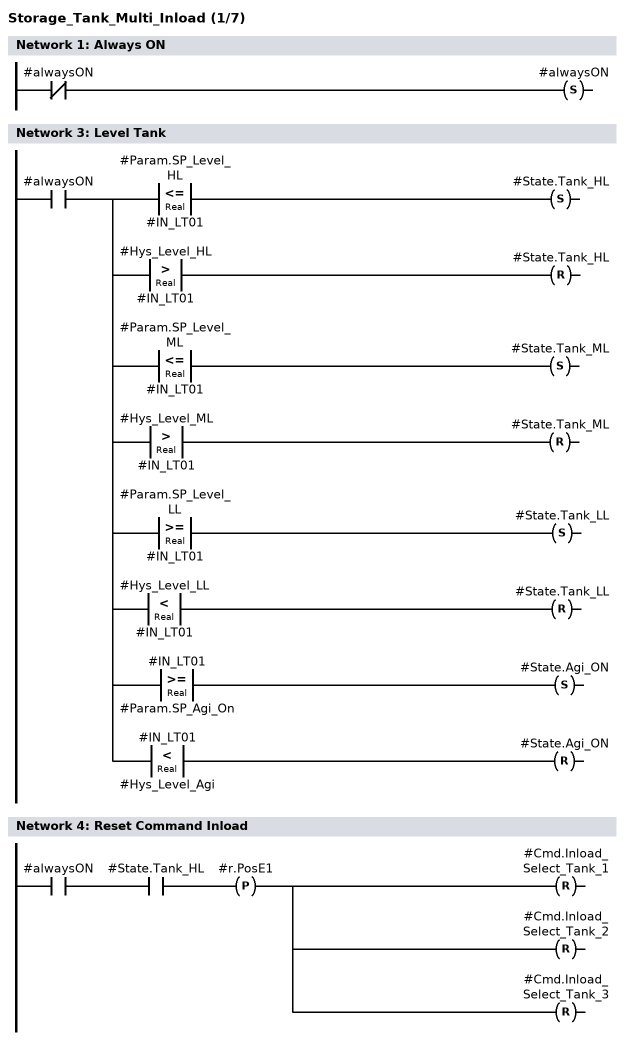
   RUNG wire#powerrail
      I_Contact( #alwaysON )
      S_Coil( #alwaysON )
   END_RUNG
   // the same network as SCL:
   IF NOT #alwaysON THEN #alwaysON := TRUE; END_IF;
END_REGION

NETWORK
TITLE = Hys Calculation
//Level Hys Absolute
      L     #Param.L_Hi_Lim;
      L     #Param.L_Lo_Lim;
      -R;
      L     100.0;
      /R;
      L     #Param.L_Hys;
      *R;
      T     #L_Hys_Abs;
//Tank High Level
      L     #Param.SP_Level_HL;
      L     #L_Hys_Abs;
      -R;
      T     #Hys_Level_HL;
//Tank Mid Level
      L     #Param.SP_Level_ML;
      L     #L_Hys_Abs;
      -R;
      T     #Hys_Level_ML;
//Tank Low Level
      L     #Param.SP_Level_LL;
      L     #L_Hys_Abs;
      +R;
      T     #Hys_Level_LL;
//Level Agi On
      L     #Param.SP_Agi_On;
      L     #L_Hys_Abs;
      -R;
      T     #Hys_Level_Agi;




REGION Network 3: Level Tank
   RUNG wire#powerrail
      Contact( #alwaysON )
      wire#w1
      { S7_Templates := "SrcType := Real" } LE_Contact(in1 := #Param.SP_Level_HL, in2 := #IN_LT01)
      S_Coil( #State.Tank_HL )
   END_RUNG
   RUNG wire#w1
      { S7_Templates := "SrcType := Real" } GT_Contact(in1 := #Hys_Level_HL, in2 := #IN_LT01)
      R_Coil( #State.Tank_HL )
   END_RUNG
   RUNG wire#w1
      { S7_Templates := "SrcType := Real" } LE_Contact(in1 := #Param.SP_Level_ML, in2 := #IN_LT01)
      S_Coil( #State.Tank_ML )
   END_RUNG
   RUNG wire#w1
      { S7_Templates := "SrcType := Real" } GT_Contact(in1 := #Hys_Level_ML, in2 := #IN_LT01)
      R_Coil( #State.Tank_ML )
   END_RUNG
   RUNG wire#w1
      { S7_Templates := "SrcType := Real" } GE_Contact(in1 := #Param.SP_Level_LL, in2 := #IN_LT01)
      S_Coil( #State.Tank_LL )
   END_RUNG
   RUNG wire#w1
      { S7_Templates := "SrcType := Real" } LT_Contact(in1 := #Hys_Level_LL, in2 := #IN_LT01)
      R_Coil( #State.Tank_LL )
   END_RUNG
   RUNG wire#w1
      { S7_Templates := "SrcType := Real" } GE_Contact(in1 := #IN_LT01, in2 := #Param.SP_Agi_On)
      S_Coil( #State.Agi_ON )
   END_RUNG
   RUNG wire#w1
      { S7_Templates := "SrcType := Real" } LT_Contact(in1 := #IN_LT01, in2 := #Hys_Level_Agi)
      R_Coil( #State.Agi_ON )
   END_RUNG
   // the same network as SCL:
   IF #alwaysON AND (#Param.SP_Level_HL <= #IN_LT01) THEN #State.Tank_HL := TRUE; END_IF;
   IF #alwaysON AND (#Hys_Level_HL > #IN_LT01) THEN #State.Tank_HL := FALSE; END_IF;
   IF #alwaysON AND (#Param.SP_Level_ML <= #IN_LT01) THEN #State.Tank_ML := TRUE; END_IF;
   IF #alwaysON AND (#Hys_Level_ML > #IN_LT01) THEN #State.Tank_ML := FALSE; END_IF;
   IF #alwaysON AND (#Param.SP_Level_LL >= #IN_LT01) THEN #State.Tank_LL := TRUE; END_IF;
   IF #alwaysON AND (#Hys_Level_LL < #IN_LT01) THEN #State.Tank_LL := FALSE; END_IF;
   IF #alwaysON AND (#IN_LT01 >= #Param.SP_Agi_On) THEN #State.Agi_ON := TRUE; END_IF;
   IF #alwaysON AND (#IN_LT01 < #Hys_Level_Agi) THEN #State.Agi_ON := FALSE; END_IF;
END_REGION

REGION Network 4: Reset Command Inload
   RUNG wire#powerrail
      Contact( #alwaysON )
      Contact( #State.Tank_HL )
      P_Trig( #r.PosE1 )
      wire#w1
      R_Coil( #Cmd.Inload_Select_Tank_1 )
   END_RUNG
   RUNG wire#w1
      R_Coil( #Cmd.Inload_Select_Tank_2 )
   END_RUNG
   RUNG wire#w1
      R_Coil( #Cmd.Inload_Select_Tank_3 )
   END_RUNG
   // the same network as SCL:
   #_w1 := #alwaysON AND #State.Tank_HL;
   #_w2 := #_w1 AND NOT #r.PosE1;   // rising edge
   #r.PosE1 := #_w1;
   IF #_w2 THEN
       #Cmd.Inload_Select_Tank_1 := FALSE;
       #Cmd.Inload_Select_Tank_2 := FALSE;
       #Cmd.Inload_Select_Tank_3 := FALSE;
   END_IF;
END_REGION

REGION Network 5: Command Inload
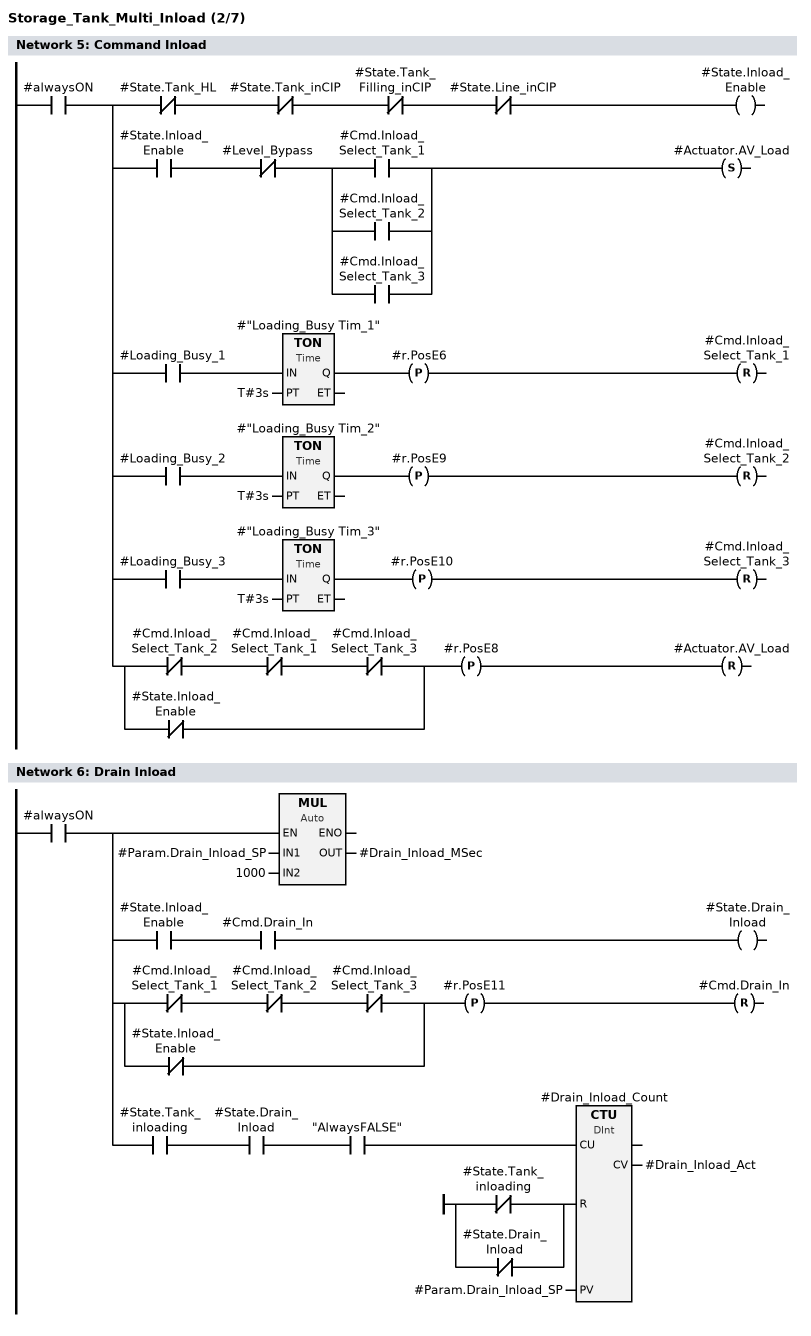
   RUNG wire#powerrail
      Contact( #alwaysON )
      wire#w1
      I_Contact( #State.Tank_HL )
      I_Contact( #State.Tank_inCIP )
      I_Contact( #State.Tank_Filling_inCIP )
      I_Contact( #State.Line_inCIP )
      Coil( #State.Inload_Enable )
   END_RUNG
   RUNG wire#w1
      Contact( #State.Inload_Enable )
      I_Contact( #Level_Bypass )
      wire#w2
      Contact( #Cmd.Inload_Select_Tank_1 )
      wire#w3
      S_Coil( #Actuator.AV_Load )
   END_RUNG
   RUNG wire#w2
      Contact( #Cmd.Inload_Select_Tank_2 )
   END_RUNG wire#w3
   RUNG wire#w2
      Contact( #Cmd.Inload_Select_Tank_3 )
   END_RUNG wire#w3
   RUNG wire#w1
      Contact( #Loading_Busy_1 )
      { S7_Templates := "time_type := Time" } #"Loading_Busy Tim_1".TON(pt := T#3s, et =>)
      P_Trig( #r.PosE6 )
      R_Coil( #Cmd.Inload_Select_Tank_1 )
   END_RUNG
   RUNG wire#w1
      Contact( #Loading_Busy_2 )
      { S7_Templates := "time_type := Time" } #"Loading_Busy Tim_2".TON(pt := T#3s, et =>)
      P_Trig( #r.PosE9 )
      R_Coil( #Cmd.Inload_Select_Tank_2 )
   END_RUNG
   RUNG wire#w1
      Contact( #Loading_Busy_3 )
      { S7_Templates := "time_type := Time" } #"Loading_Busy Tim_3".TON(pt := T#3s, et =>)
      P_Trig( #r.PosE10 )
      R_Coil( #Cmd.Inload_Select_Tank_3 )
   END_RUNG
   RUNG wire#w1
      I_Contact( #Cmd.Inload_Select_Tank_2 )
      I_Contact( #Cmd.Inload_Select_Tank_1 )
      I_Contact( #Cmd.Inload_Select_Tank_3 )
      wire#w4
      P_Trig( #r.PosE8 )
      R_Coil( #Actuator.AV_Load )
   END_RUNG
   RUNG wire#w1
      I_Contact( #State.Inload_Enable )
   END_RUNG wire#w4
   // the same network as SCL:
   #State.Inload_Enable := #alwaysON AND NOT #State.Tank_HL AND NOT #State.Tank_inCIP AND NOT #State.Tank_Filling_inCIP AND NOT #State.Line_inCIP;
   IF #alwaysON AND #State.Inload_Enable AND NOT #Level_Bypass AND (#Cmd.Inload_Select_Tank_1 OR #Cmd.Inload_Select_Tank_2 OR #Cmd.Inload_Select_Tank_3) THEN
       #Actuator.AV_Load := TRUE;
   END_IF;
   #"Loading_Busy Tim_1"(IN := #alwaysON AND #Loading_Busy_1, PT := T#3s);   // TON
   #_w1 := #"Loading_Busy Tim_1".Q AND NOT #r.PosE6;   // rising edge
   #r.PosE6 := #"Loading_Busy Tim_1".Q;
   IF #_w1 THEN #Cmd.Inload_Select_Tank_1 := FALSE; END_IF;
   #"Loading_Busy Tim_2"(IN := #alwaysON AND #Loading_Busy_2, PT := T#3s);   // TON
   #_w2 := #"Loading_Busy Tim_2".Q AND NOT #r.PosE9;   // rising edge
   #r.PosE9 := #"Loading_Busy Tim_2".Q;
   IF #_w2 THEN #Cmd.Inload_Select_Tank_2 := FALSE; END_IF;
   #"Loading_Busy Tim_3"(IN := #alwaysON AND #Loading_Busy_3, PT := T#3s);   // TON
   #_w3 := #"Loading_Busy Tim_3".Q AND NOT #r.PosE10;   // rising edge
   #r.PosE10 := #"Loading_Busy Tim_3".Q;
   IF #_w3 THEN #Cmd.Inload_Select_Tank_3 := FALSE; END_IF;
   #_w4 := #alwaysON AND ((NOT #Cmd.Inload_Select_Tank_2 AND NOT #Cmd.Inload_Select_Tank_1 AND NOT #Cmd.Inload_Select_Tank_3) OR NOT #State.Inload_Enable);
   #_w5 := #_w4 AND NOT #r.PosE8;   // rising edge
   #r.PosE8 := #_w4;
   IF #_w5 THEN #Actuator.AV_Load := FALSE; END_IF;
END_REGION

REGION Network 6: Drain Inload
   RUNG wire#powerrail
      Contact( #alwaysON )
      wire#w1
      Mul(in1 := #Param.Drain_Inload_SP, in2 := 1000, out => #Drain_Inload_MSec)
   END_RUNG
   RUNG wire#w1
      Contact( #State.Inload_Enable )
      Contact( #Cmd.Drain_In )
      Coil( #State.Drain_Inload )
   END_RUNG
   RUNG wire#w1
      I_Contact( #Cmd.Inload_Select_Tank_1 )
      I_Contact( #Cmd.Inload_Select_Tank_2 )
      I_Contact( #Cmd.Inload_Select_Tank_3 )
      wire#w2
      P_Trig( #r.PosE11 )
      R_Coil( #Cmd.Drain_In )
   END_RUNG
   RUNG wire#w1
      I_Contact( #State.Inload_Enable )
   END_RUNG wire#w2
   RUNG wire#w1
      Contact( #State.Tank_inloading )
      Contact( #State.Drain_Inload )
      Contact( "AlwaysFALSE" )
      { S7_Templates := "value_type := DInt" } #Drain_Inload_Count.CTU(r := wire#w3, pv := #Param.Drain_Inload_SP, cv => #Drain_Inload_Act)
   END_RUNG
   RUNG wire#powerrail
      I_Contact( #State.Tank_inloading )
   END_RUNG wire#w3
   RUNG wire#powerrail
      I_Contact( #State.Drain_Inload )
   END_RUNG wire#w3
   // the same network as SCL:
   IF #alwaysON THEN #Drain_Inload_MSec := #Param.Drain_Inload_SP * 1000; END_IF;
   #State.Drain_Inload := #alwaysON AND #State.Inload_Enable AND #Cmd.Drain_In;
   #_w1 := #alwaysON AND ((NOT #Cmd.Inload_Select_Tank_1 AND NOT #Cmd.Inload_Select_Tank_2 AND NOT #Cmd.Inload_Select_Tank_3) OR NOT #State.Inload_Enable);
   #_w2 := #_w1 AND NOT #r.PosE11;   // rising edge
   #r.PosE11 := #_w1;
   IF #_w2 THEN #Cmd.Drain_In := FALSE; END_IF;
   #Drain_Inload_Count.CTU(CU := #alwaysON AND #State.Tank_inloading AND #State.Drain_Inload AND "AlwaysFALSE",
                           R := NOT #State.Tank_inloading OR NOT #State.Drain_Inload,
                           PV := #Param.Drain_Inload_SP,
                           CV => #Drain_Inload_Act);
END_REGION

REGION Network 7: Command Transfer to Filling
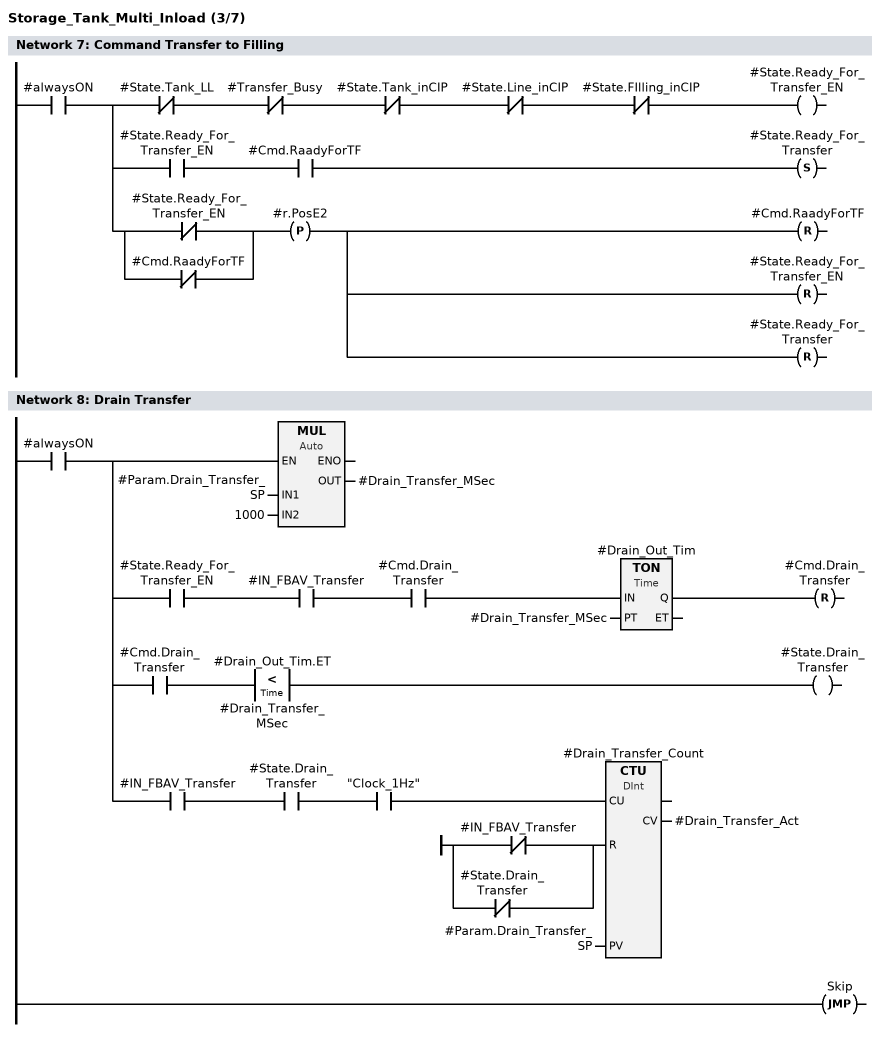
   RUNG wire#powerrail
      Contact( #alwaysON )
      wire#w1
      I_Contact( #State.Tank_LL )
      I_Contact( #Transfer_Busy )
      I_Contact( #State.Tank_inCIP )
      I_Contact( #State.Line_inCIP )
      I_Contact( #State.FIlling_inCIP )
      Coil( #State.Ready_For_Transfer_EN )
   END_RUNG
   RUNG wire#w1
      Contact( #State.Ready_For_Transfer_EN )
      Contact( #Cmd.RaadyForTF )
      S_Coil( #State.Ready_For_Transfer )
   END_RUNG
   RUNG wire#w1
      I_Contact( #State.Ready_For_Transfer_EN )
      wire#w2
      P_Trig( #r.PosE2 )
      wire#w3
      R_Coil( #Cmd.RaadyForTF )
   END_RUNG
   RUNG wire#w1
      I_Contact( #Cmd.RaadyForTF )
   END_RUNG wire#w2
   RUNG wire#w3
      R_Coil( #State.Ready_For_Transfer_EN )
   END_RUNG
   RUNG wire#w3
      R_Coil( #State.Ready_For_Transfer )
   END_RUNG
   // the same network as SCL:
   #State.Ready_For_Transfer_EN := #alwaysON AND NOT #State.Tank_LL AND NOT #Transfer_Busy AND NOT #State.Tank_inCIP AND NOT #State.Line_inCIP AND NOT #State.FIlling_inCIP;
   IF #alwaysON AND #State.Ready_For_Transfer_EN AND #Cmd.RaadyForTF THEN
       #State.Ready_For_Transfer := TRUE;
   END_IF;
   #_w1 := #alwaysON AND (NOT #State.Ready_For_Transfer_EN OR NOT #Cmd.RaadyForTF);
   #_w2 := #_w1 AND NOT #r.PosE2;   // rising edge
   #r.PosE2 := #_w1;
   IF #_w2 THEN
       #Cmd.RaadyForTF := FALSE;
       #State.Ready_For_Transfer_EN := FALSE;
       #State.Ready_For_Transfer := FALSE;
   END_IF;
END_REGION

REGION Network 8: Drain Transfer
   RUNG wire#powerrail
      Contact( #alwaysON )
      wire#w1
      Mul(in1 := #Param.Drain_Transfer_SP, in2 := 1000, out => #Drain_Transfer_MSec)
   END_RUNG
   RUNG wire#w1
      Contact( #State.Ready_For_Transfer_EN )
      Contact( #IN_FBAV_Transfer )
      Contact( #Cmd.Drain_Transfer )
      { S7_Templates := "time_type := Time" } #Drain_Out_Tim.TON(pt := #Drain_Transfer_MSec, et =>)
      R_Coil( #Cmd.Drain_Transfer )
   END_RUNG
   RUNG wire#w1
      Contact( #Cmd.Drain_Transfer )
      { S7_Templates := "SrcType := Time" } LT_Contact(in1 := #Drain_Out_Tim.ET, in2 := #Drain_Transfer_MSec)
      Coil( #State.Drain_Transfer )
   END_RUNG
   RUNG wire#w1
      Contact( #IN_FBAV_Transfer )
      Contact( #State.Drain_Transfer )
      Contact( "Clock_1Hz" )
      { S7_Templates := "value_type := DInt" } #Drain_Transfer_Count.CTU(r := wire#w2, pv := #Param.Drain_Transfer_SP, cv => #Drain_Transfer_Act)
   END_RUNG
   RUNG wire#powerrail
      I_Contact( #IN_FBAV_Transfer )
   END_RUNG wire#w2
   RUNG wire#powerrail
      I_Contact( #State.Drain_Transfer )
   END_RUNG wire#w2
   RUNG wire#powerrail
      JumpCoil( Skip )
   END_RUNG
   // the same network as SCL:
   IF #alwaysON THEN #Drain_Transfer_MSec := #Param.Drain_Transfer_SP * 1000; END_IF;
   #Drain_Out_Tim(IN := #alwaysON AND #State.Ready_For_Transfer_EN AND #IN_FBAV_Transfer AND #Cmd.Drain_Transfer,   // TON
                  PT := #Drain_Transfer_MSec);
   IF #Drain_Out_Tim.Q THEN #Cmd.Drain_Transfer := FALSE; END_IF;
   #State.Drain_Transfer := #alwaysON AND #Cmd.Drain_Transfer AND (#Drain_Out_Tim.ET < #Drain_Transfer_MSec);
   #Drain_Transfer_Count.CTU(CU := #alwaysON AND #IN_FBAV_Transfer AND #State.Drain_Transfer AND "Clock_1Hz",
                           R := NOT #IN_FBAV_Transfer OR NOT #State.Drain_Transfer,
                           PV := #Param.Drain_Transfer_SP,
                           CV => #Drain_Transfer_Act);
   GOTO Skip;
END_REGION

REGION Network 9: -----------------------------------------------State transfer to filling
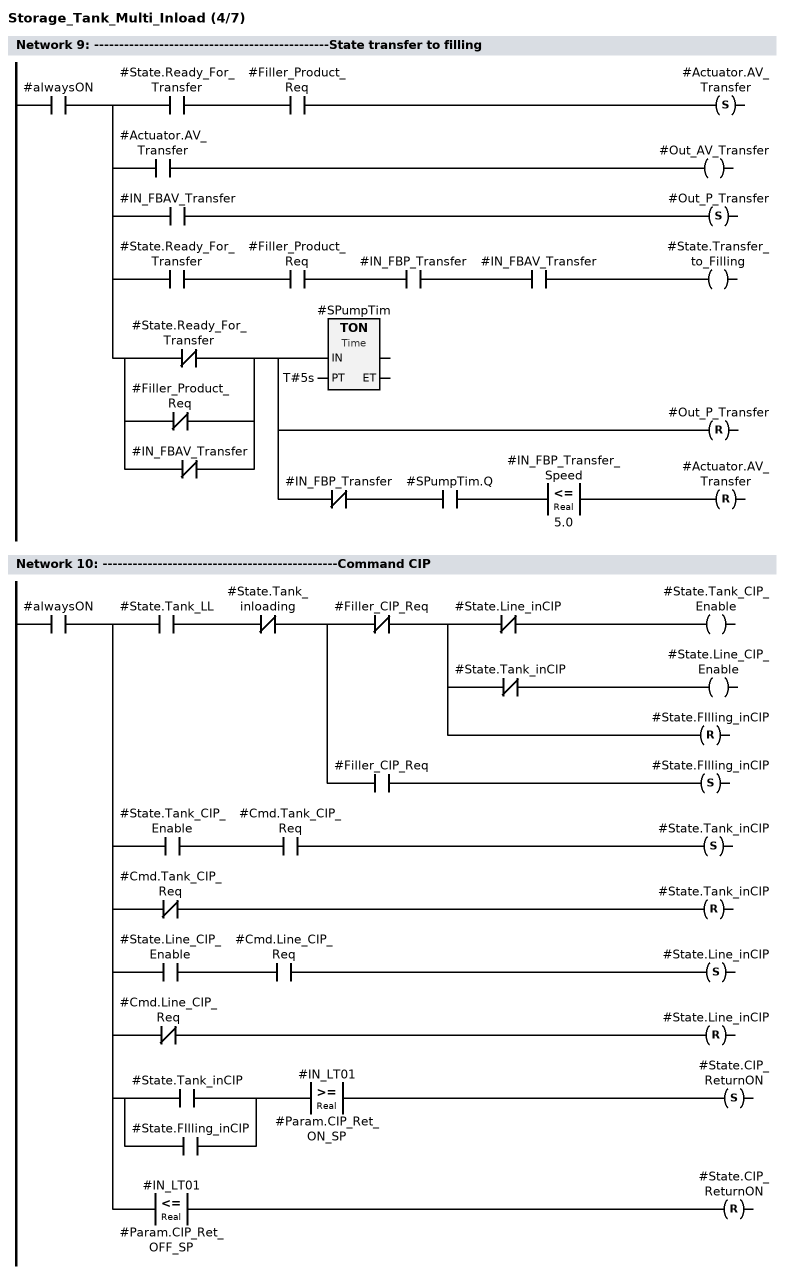
   RUNG wire#powerrail
      Contact( #alwaysON )
      wire#w1
      Contact( #State.Ready_For_Transfer )
      Contact( #Filler_Product_Req )
      S_Coil( #Actuator.AV_Transfer )
   END_RUNG
   RUNG wire#w1
      Contact( #Actuator.AV_Transfer )
      Coil( #Out_AV_Transfer )
   END_RUNG
   RUNG wire#w1
      Contact( #IN_FBAV_Transfer )
      S_Coil( #Out_P_Transfer )
   END_RUNG
   RUNG wire#w1
      Contact( #State.Ready_For_Transfer )
      Contact( #Filler_Product_Req )
      Contact( #IN_FBP_Transfer )
      Contact( #IN_FBAV_Transfer )
      Coil( #State.Transfer_to_Filling )
   END_RUNG
   RUNG wire#w1
      I_Contact( #State.Ready_For_Transfer )
      wire#w2
      { S7_Templates := "time_type := Time" } #SPumpTim.TON(pt := T#5s, et =>)
   END_RUNG
   RUNG wire#w1
      I_Contact( #Filler_Product_Req )
   END_RUNG wire#w2
   RUNG wire#w1
      I_Contact( #IN_FBAV_Transfer )
   END_RUNG wire#w2
   RUNG wire#w2
      R_Coil( #Out_P_Transfer )
   END_RUNG
   RUNG wire#w2
      I_Contact( #IN_FBP_Transfer )
      Contact( #SPumpTim.Q )
      { S7_Templates := "SrcType := Real" } LE_Contact(in1 := #IN_FBP_Transfer_Speed, in2 := 5.0)
      R_Coil( #Actuator.AV_Transfer )
   END_RUNG
   // the same network as SCL:
   IF #alwaysON AND #State.Ready_For_Transfer AND #Filler_Product_Req THEN
       #Actuator.AV_Transfer := TRUE;
   END_IF;
   #Out_AV_Transfer := #alwaysON AND #Actuator.AV_Transfer;
   IF #alwaysON AND #IN_FBAV_Transfer THEN #Out_P_Transfer := TRUE; END_IF;
   #State.Transfer_to_Filling := #alwaysON AND #State.Ready_For_Transfer AND #Filler_Product_Req AND #IN_FBP_Transfer AND #IN_FBAV_Transfer;
   #_w1 := #alwaysON AND (NOT #State.Ready_For_Transfer OR NOT #Filler_Product_Req OR NOT #IN_FBAV_Transfer);
   #SPumpTim(IN := #_w1, PT := T#5s);   // TON
   IF #_w1 THEN #Out_P_Transfer := FALSE; END_IF;
   IF #_w1 AND NOT #IN_FBP_Transfer AND #SPumpTim.Q AND (#IN_FBP_Transfer_Speed <= 5.0) THEN
       #Actuator.AV_Transfer := FALSE;
   END_IF;
END_REGION

REGION Network 10: -----------------------------------------------Command CIP
   RUNG wire#powerrail
      Contact( #alwaysON )
      wire#w1
      Contact( #State.Tank_LL )
      I_Contact( #State.Tank_inloading )
      wire#w2
      I_Contact( #Filler_CIP_Req )
      wire#w3
      I_Contact( #State.Line_inCIP )
      Coil( #State.Tank_CIP_Enable )
   END_RUNG
   RUNG wire#w3
      I_Contact( #State.Tank_inCIP )
      Coil( #State.Line_CIP_Enable )
   END_RUNG
   RUNG wire#w3
      R_Coil( #State.FIlling_inCIP )
   END_RUNG
   RUNG wire#w2
      Contact( #Filler_CIP_Req )
      S_Coil( #State.FIlling_inCIP )
   END_RUNG
   RUNG wire#w1
      Contact( #State.Tank_CIP_Enable )
      Contact( #Cmd.Tank_CIP_Req )
      S_Coil( #State.Tank_inCIP )
   END_RUNG
   RUNG wire#w1
      I_Contact( #Cmd.Tank_CIP_Req )
      R_Coil( #State.Tank_inCIP )
   END_RUNG
   RUNG wire#w1
      Contact( #State.Line_CIP_Enable )
      Contact( #Cmd.Line_CIP_Req )
      S_Coil( #State.Line_inCIP )
   END_RUNG
   RUNG wire#w1
      I_Contact( #Cmd.Line_CIP_Req )
      R_Coil( #State.Line_inCIP )
   END_RUNG
   RUNG wire#w1
      Contact( #State.Tank_inCIP )
      wire#w4
      { S7_Templates := "SrcType := Real" } GE_Contact(in1 := #IN_LT01, in2 := #Param.CIP_Ret_ON_SP)
      S_Coil( #State.CIP_ReturnON )
   END_RUNG
   RUNG wire#w1
      Contact( #State.FIlling_inCIP )
   END_RUNG wire#w4
   RUNG wire#w1
      { S7_Templates := "SrcType := Real" } LE_Contact(in1 := #IN_LT01, in2 := #Param.CIP_Ret_OFF_SP)
      R_Coil( #State.CIP_ReturnON )
   END_RUNG
   // the same network as SCL:
   #_w1 := #alwaysON AND #State.Tank_LL AND NOT #State.Tank_inloading;
   #_w2 := #_w1 AND NOT #Filler_CIP_Req;
   #State.Tank_CIP_Enable := #_w2 AND NOT #State.Line_inCIP;
   #State.Line_CIP_Enable := #_w2 AND NOT #State.Tank_inCIP;
   IF #_w2 THEN #State.FIlling_inCIP := FALSE; END_IF;
   IF #_w1 AND #Filler_CIP_Req THEN #State.FIlling_inCIP := TRUE; END_IF;
   IF #alwaysON AND #State.Tank_CIP_Enable AND #Cmd.Tank_CIP_Req THEN #State.Tank_inCIP := TRUE; END_IF;
   IF #alwaysON AND NOT #Cmd.Tank_CIP_Req THEN #State.Tank_inCIP := FALSE; END_IF;
   IF #alwaysON AND #State.Line_CIP_Enable AND #Cmd.Line_CIP_Req THEN #State.Line_inCIP := TRUE; END_IF;
   IF #alwaysON AND NOT #Cmd.Line_CIP_Req THEN #State.Line_inCIP := FALSE; END_IF;
   IF #alwaysON AND (#State.Tank_inCIP OR #State.FIlling_inCIP) AND (#IN_LT01 >= #Param.CIP_Ret_ON_SP) THEN
       #State.CIP_ReturnON := TRUE;
   END_IF;
   IF #alwaysON AND (#IN_LT01 <= #Param.CIP_Ret_OFF_SP) THEN #State.CIP_ReturnON := FALSE; END_IF;
END_REGION

REGION Network 11: Command CIP New
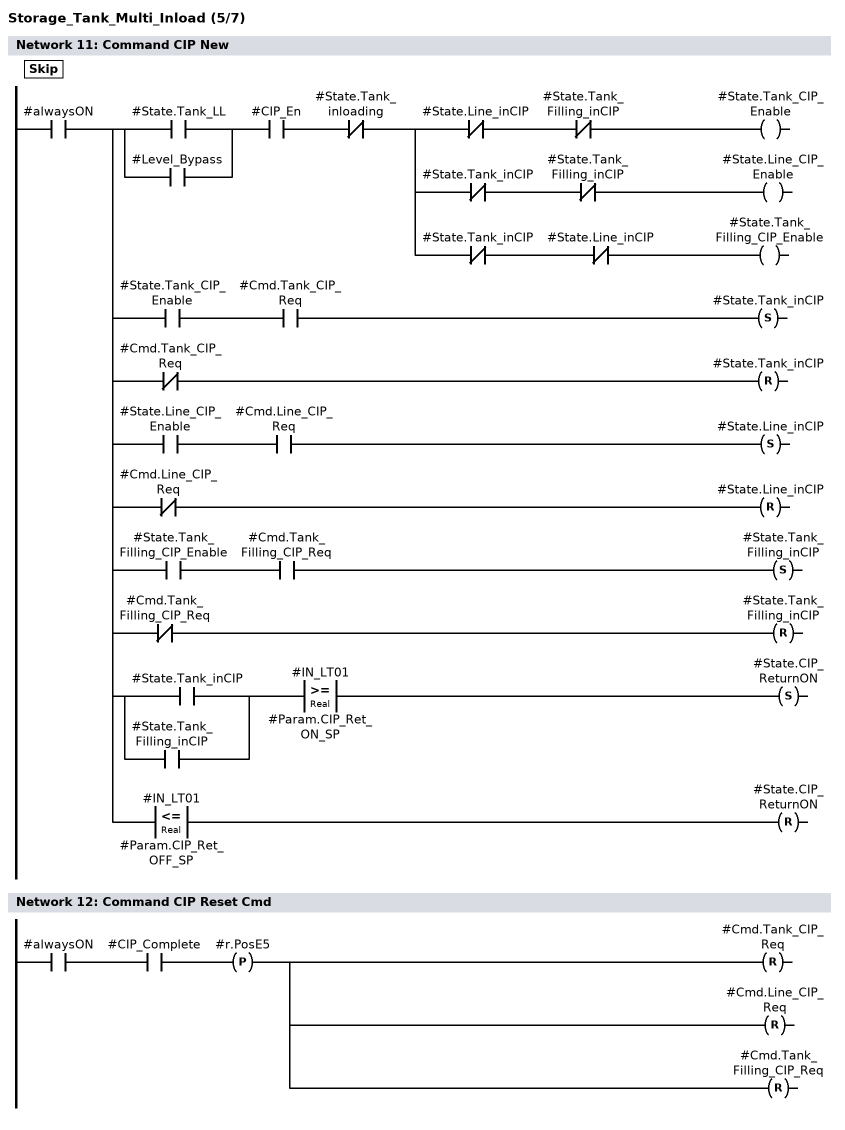
   Label( Skip )
   RUNG wire#powerrail
      Contact( #alwaysON )
      wire#w1
      Contact( #State.Tank_LL )
      wire#w2
      Contact( #CIP_En )
      I_Contact( #State.Tank_inloading )
      wire#w3
      I_Contact( #State.Line_inCIP )
      I_Contact( #State.Tank_Filling_inCIP )
      Coil( #State.Tank_CIP_Enable )
   END_RUNG
   RUNG wire#w1
      Contact( #Level_Bypass )
   END_RUNG wire#w2
   RUNG wire#w3
      I_Contact( #State.Tank_inCIP )
      I_Contact( #State.Tank_Filling_inCIP )
      Coil( #State.Line_CIP_Enable )
   END_RUNG
   RUNG wire#w3
      I_Contact( #State.Tank_inCIP )
      I_Contact( #State.Line_inCIP )
      Coil( #State.Tank_Filling_CIP_Enable )
   END_RUNG
   RUNG wire#w1
      Contact( #State.Tank_CIP_Enable )
      Contact( #Cmd.Tank_CIP_Req )
      S_Coil( #State.Tank_inCIP )
   END_RUNG
   RUNG wire#w1
      I_Contact( #Cmd.Tank_CIP_Req )
      R_Coil( #State.Tank_inCIP )
   END_RUNG
   RUNG wire#w1
      Contact( #State.Line_CIP_Enable )
      Contact( #Cmd.Line_CIP_Req )
      S_Coil( #State.Line_inCIP )
   END_RUNG
   RUNG wire#w1
      I_Contact( #Cmd.Line_CIP_Req )
      R_Coil( #State.Line_inCIP )
   END_RUNG
   RUNG wire#w1
      Contact( #State.Tank_Filling_CIP_Enable )
      Contact( #Cmd.Tank_Filling_CIP_Req )
      S_Coil( #State.Tank_Filling_inCIP )
   END_RUNG
   RUNG wire#w1
      I_Contact( #Cmd.Tank_Filling_CIP_Req )
      R_Coil( #State.Tank_Filling_inCIP )
   END_RUNG
   RUNG wire#w1
      Contact( #State.Tank_inCIP )
      wire#w4
      { S7_Templates := "SrcType := Real" } GE_Contact(in1 := #IN_LT01, in2 := #Param.CIP_Ret_ON_SP)
      S_Coil( #State.CIP_ReturnON )
   END_RUNG
   RUNG wire#w1
      Contact( #State.Tank_Filling_inCIP )
   END_RUNG wire#w4
   RUNG wire#w1
      { S7_Templates := "SrcType := Real" } LE_Contact(in1 := #IN_LT01, in2 := #Param.CIP_Ret_OFF_SP)
      R_Coil( #State.CIP_ReturnON )
   END_RUNG
   // the same network as SCL:
   Skip:
   #_w1 := #alwaysON AND (#State.Tank_LL OR #Level_Bypass) AND #CIP_En AND NOT #State.Tank_inloading;
   #State.Tank_CIP_Enable := #_w1 AND NOT #State.Line_inCIP AND NOT #State.Tank_Filling_inCIP;
   #State.Line_CIP_Enable := #_w1 AND NOT #State.Tank_inCIP AND NOT #State.Tank_Filling_inCIP;
   #State.Tank_Filling_CIP_Enable := #_w1 AND NOT #State.Tank_inCIP AND NOT #State.Line_inCIP;
   IF #alwaysON AND #State.Tank_CIP_Enable AND #Cmd.Tank_CIP_Req THEN #State.Tank_inCIP := TRUE; END_IF;
   IF #alwaysON AND NOT #Cmd.Tank_CIP_Req THEN #State.Tank_inCIP := FALSE; END_IF;
   IF #alwaysON AND #State.Line_CIP_Enable AND #Cmd.Line_CIP_Req THEN #State.Line_inCIP := TRUE; END_IF;
   IF #alwaysON AND NOT #Cmd.Line_CIP_Req THEN #State.Line_inCIP := FALSE; END_IF;
   IF #alwaysON AND #State.Tank_Filling_CIP_Enable AND #Cmd.Tank_Filling_CIP_Req THEN
       #State.Tank_Filling_inCIP := TRUE;
   END_IF;
   IF #alwaysON AND NOT #Cmd.Tank_Filling_CIP_Req THEN #State.Tank_Filling_inCIP := FALSE; END_IF;
   IF #alwaysON AND (#State.Tank_inCIP OR #State.Tank_Filling_inCIP) AND (#IN_LT01 >= #Param.CIP_Ret_ON_SP) THEN
       #State.CIP_ReturnON := TRUE;
   END_IF;
   IF #alwaysON AND (#IN_LT01 <= #Param.CIP_Ret_OFF_SP) THEN #State.CIP_ReturnON := FALSE; END_IF;
END_REGION

REGION Network 12: Command CIP Reset Cmd
   RUNG wire#powerrail
      Contact( #alwaysON )
      Contact( #CIP_Complete )
      P_Trig( #r.PosE5 )
      wire#w1
      R_Coil( #Cmd.Tank_CIP_Req )
   END_RUNG
   RUNG wire#w1
      R_Coil( #Cmd.Line_CIP_Req )
   END_RUNG
   RUNG wire#w1
      R_Coil( #Cmd.Tank_Filling_CIP_Req )
   END_RUNG
   // the same network as SCL:
   #_w1 := #alwaysON AND #CIP_Complete;
   #_w2 := #_w1 AND NOT #r.PosE5;   // rising edge
   #r.PosE5 := #_w1;
   IF #_w2 THEN
       #Cmd.Tank_CIP_Req := FALSE;
       #Cmd.Line_CIP_Req := FALSE;
       #Cmd.Tank_Filling_CIP_Req := FALSE;
   END_IF;
END_REGION

REGION Network 13: Send CIP Request
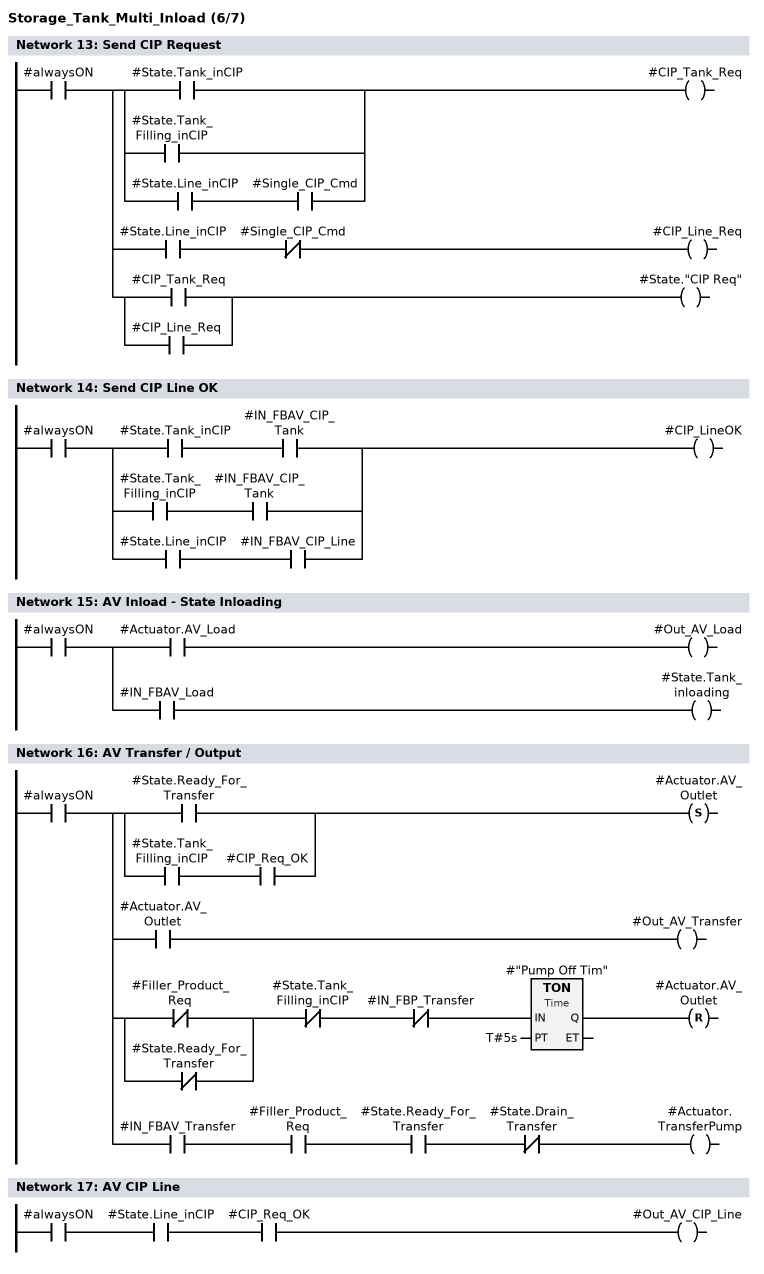
   RUNG wire#powerrail
      Contact( #alwaysON )
      wire#w1
      Contact( #State.Tank_inCIP )
      wire#w2
      Coil( #CIP_Tank_Req )
   END_RUNG
   RUNG wire#w1
      Contact( #State.Tank_Filling_inCIP )
   END_RUNG wire#w2
   RUNG wire#w1
      Contact( #State.Line_inCIP )
      Contact( #Single_CIP_Cmd )
   END_RUNG wire#w2
   RUNG wire#w1
      Contact( #State.Line_inCIP )
      I_Contact( #Single_CIP_Cmd )
      Coil( #CIP_Line_Req )
   END_RUNG
   RUNG wire#w1
      Contact( #CIP_Tank_Req )
      wire#w3
      Coil( #State."CIP Req" )
   END_RUNG
   RUNG wire#w1
      Contact( #CIP_Line_Req )
   END_RUNG wire#w3
   // the same network as SCL:
   #CIP_Tank_Req := #alwaysON AND (#State.Tank_inCIP OR #State.Tank_Filling_inCIP OR (#State.Line_inCIP AND #Single_CIP_Cmd));
   #CIP_Line_Req := #alwaysON AND #State.Line_inCIP AND NOT #Single_CIP_Cmd;
   #State."CIP Req" := #alwaysON AND (#CIP_Tank_Req OR #CIP_Line_Req);
END_REGION

REGION Network 14: Send CIP Line OK
   RUNG wire#powerrail
      Contact( #alwaysON )
      wire#w1
      Contact( #State.Tank_inCIP )
      Contact( #IN_FBAV_CIP_Tank )
      wire#w2
      Coil( #CIP_LineOK )
   END_RUNG
   RUNG wire#w1
      Contact( #State.Tank_Filling_inCIP )
      Contact( #IN_FBAV_CIP_Tank )
   END_RUNG wire#w2
   RUNG wire#w1
      Contact( #State.Line_inCIP )
      Contact( #IN_FBAV_CIP_Line )
   END_RUNG wire#w2
   // the same network as SCL:
   #CIP_LineOK := #alwaysON AND ((#State.Tank_inCIP AND #IN_FBAV_CIP_Tank) OR (#State.Tank_Filling_inCIP AND #IN_FBAV_CIP_Tank) OR (#State.Line_inCIP AND #IN_FBAV_CIP_Line));
END_REGION

REGION Network 15: AV Inload - State Inloading
   RUNG wire#powerrail
      Contact( #alwaysON )
      wire#w1
      Contact( #Actuator.AV_Load )
      Coil( #Out_AV_Load )
   END_RUNG
   RUNG wire#w1
      Contact( #IN_FBAV_Load )
      Coil( #State.Tank_inloading )
   END_RUNG
   // the same network as SCL:
   #Out_AV_Load := #alwaysON AND #Actuator.AV_Load;
   #State.Tank_inloading := #alwaysON AND #IN_FBAV_Load;
END_REGION

REGION Network 16: AV Transfer / Output
   RUNG wire#powerrail
      Contact( #alwaysON )
      wire#w1
      Contact( #State.Ready_For_Transfer )
      wire#w2
      S_Coil( #Actuator.AV_Outlet )
   END_RUNG
   RUNG wire#w1
      Contact( #State.Tank_Filling_inCIP )
      Contact( #CIP_Req_OK )
   END_RUNG wire#w2
   RUNG wire#w1
      Contact( #Actuator.AV_Outlet )
      Coil( #Out_AV_Transfer )
   END_RUNG
   RUNG wire#w1
      I_Contact( #Filler_Product_Req )
      wire#w3
      I_Contact( #State.Tank_Filling_inCIP )
      I_Contact( #IN_FBP_Transfer )
      { S7_Templates := "time_type := Time" } #"Pump Off Tim".TON(pt := T#5s, et =>)
      R_Coil( #Actuator.AV_Outlet )
   END_RUNG
   RUNG wire#w1
      I_Contact( #State.Ready_For_Transfer )
   END_RUNG wire#w3
   RUNG wire#w1
      Contact( #IN_FBAV_Transfer )
      Contact( #Filler_Product_Req )
      Contact( #State.Ready_For_Transfer )
      I_Contact( #State.Drain_Transfer )
      Coil( #Actuator.TransferPump )
   END_RUNG
   // the same network as SCL:
   IF #alwaysON AND (#State.Ready_For_Transfer OR (#State.Tank_Filling_inCIP AND #CIP_Req_OK)) THEN
       #Actuator.AV_Outlet := TRUE;
   END_IF;
   #Out_AV_Transfer := #alwaysON AND #Actuator.AV_Outlet;
   #"Pump Off Tim"(IN := #alwaysON AND (NOT #Filler_Product_Req OR NOT #State.Ready_For_Transfer) AND NOT #State.Tank_Filling_inCIP AND NOT #IN_FBP_Transfer,   // TON
                   PT := T#5s);
   IF #"Pump Off Tim".Q THEN #Actuator.AV_Outlet := FALSE; END_IF;
   #Actuator.TransferPump := #alwaysON AND #IN_FBAV_Transfer AND #Filler_Product_Req AND #State.Ready_For_Transfer AND NOT #State.Drain_Transfer;
END_REGION

REGION Network 17: AV CIP Line
   RUNG wire#powerrail
      Contact( #alwaysON )
      Contact( #State.Line_inCIP )
      Contact( #CIP_Req_OK )
      Coil( #Out_AV_CIP_Line )
   END_RUNG
   // the same network as SCL:
   #Out_AV_CIP_Line := #alwaysON AND #State.Line_inCIP AND #CIP_Req_OK;
END_REGION

REGION Network 18: AV CIP Tank to Filling
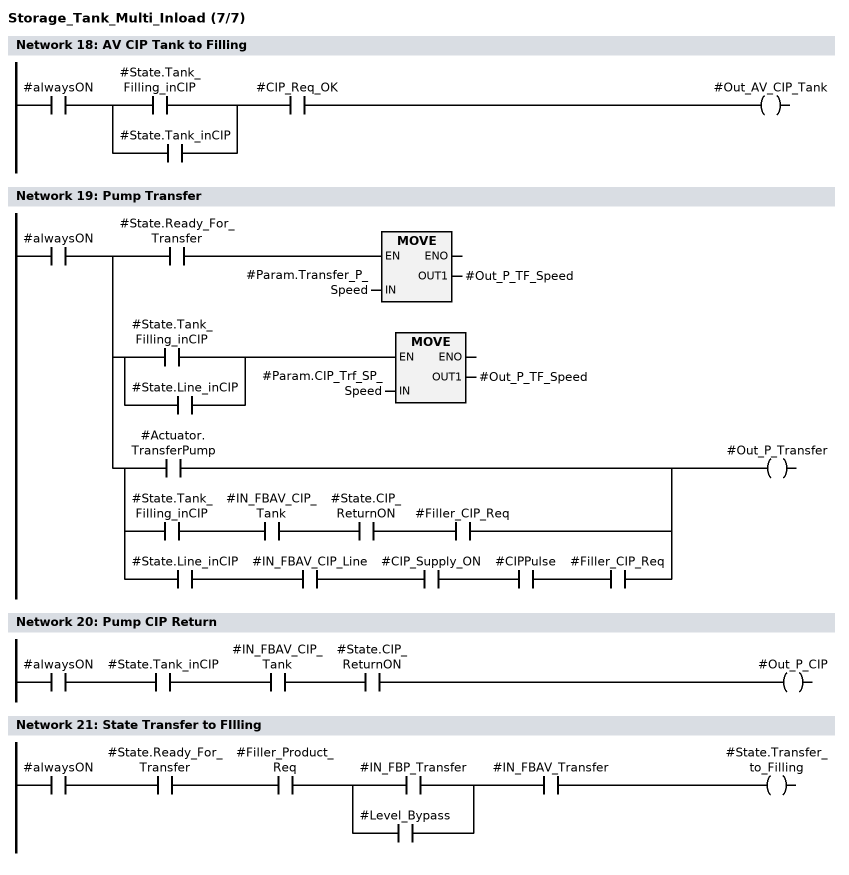
   RUNG wire#powerrail
      Contact( #alwaysON )
      wire#w1
      Contact( #State.Tank_Filling_inCIP )
      wire#w2
      Contact( #CIP_Req_OK )
      Coil( #Out_AV_CIP_Tank )
   END_RUNG
   RUNG wire#w1
      Contact( #State.Tank_inCIP )
   END_RUNG wire#w2
   // the same network as SCL:
   #Out_AV_CIP_Tank := #alwaysON AND (#State.Tank_Filling_inCIP OR #State.Tank_inCIP) AND #CIP_Req_OK;
END_REGION

REGION Network 19: Pump Transfer
   RUNG wire#powerrail
      Contact( #alwaysON )
      wire#w1
      Contact( #State.Ready_For_Transfer )
      Move(in := #Param.Transfer_P_Speed, out1 => #Out_P_TF_Speed)
   END_RUNG
   RUNG wire#w1
      Contact( #State.Tank_Filling_inCIP )
      wire#w2
      Move(in := #Param.CIP_Trf_SP_Speed, out1 => #Out_P_TF_Speed)
   END_RUNG
   RUNG wire#w1
      Contact( #State.Line_inCIP )
   END_RUNG wire#w2
   RUNG wire#w1
      Contact( #Actuator.TransferPump )
      wire#w3
      Coil( #Out_P_Transfer )
   END_RUNG
   RUNG wire#w1
      Contact( #State.Tank_Filling_inCIP )
      Contact( #IN_FBAV_CIP_Tank )
      Contact( #State.CIP_ReturnON )
      Contact( #Filler_CIP_Req )
   END_RUNG wire#w3
   RUNG wire#w1
      Contact( #State.Line_inCIP )
      Contact( #IN_FBAV_CIP_Line )
      Contact( #CIP_Supply_ON )
      Contact( #CIPPulse )
      Contact( #Filler_CIP_Req )
   END_RUNG wire#w3
   // the same network as SCL:
   IF #alwaysON AND #State.Ready_For_Transfer THEN #Out_P_TF_Speed := #Param.Transfer_P_Speed; END_IF;
   IF #alwaysON AND (#State.Tank_Filling_inCIP OR #State.Line_inCIP) THEN
       #Out_P_TF_Speed := #Param.CIP_Trf_SP_Speed;
   END_IF;
   #Out_P_Transfer := #alwaysON AND (#Actuator.TransferPump OR (#State.Tank_Filling_inCIP AND #IN_FBAV_CIP_Tank AND #State.CIP_ReturnON AND #Filler_CIP_Req) OR (#State.Line_inCIP AND #IN_FBAV_CIP_Line AND #CIP_Supply_ON AND #CIPPulse AND #Filler_CIP_Req));
END_REGION

REGION Network 20: Pump CIP Return
   RUNG wire#powerrail
      Contact( #alwaysON )
      Contact( #State.Tank_inCIP )
      Contact( #IN_FBAV_CIP_Tank )
      Contact( #State.CIP_ReturnON )
      Coil( #Out_P_CIP )
   END_RUNG
   // the same network as SCL:
   #Out_P_CIP := #alwaysON AND #State.Tank_inCIP AND #IN_FBAV_CIP_Tank AND #State.CIP_ReturnON;
END_REGION

REGION Network 21: State Transfer to FIlling
   RUNG wire#powerrail
      Contact( #alwaysON )
      Contact( #State.Ready_For_Transfer )
      Contact( #Filler_Product_Req )
      wire#w1
      Contact( #IN_FBP_Transfer )
      wire#w2
      Contact( #IN_FBAV_Transfer )
      Coil( #State.Transfer_to_Filling )
   END_RUNG
   RUNG wire#w1
      Contact( #Level_Bypass )
   END_RUNG wire#w2
   // the same network as SCL:
   #State.Transfer_to_Filling := #alwaysON AND #State.Ready_For_Transfer AND #Filler_Product_Req AND (#IN_FBP_Transfer OR #Level_Bypass) AND #IN_FBAV_Transfer;
END_REGION
END_FUNCTION_BLOCK

FUNCTION "Buffer" : Void   // FC11, LAD
{ S7_Optimized_Access := 'TRUE' }
VERSION : 0.1
// stored: AutoNumber true, IsIECCheckEnabled false, SetENOAutomatically false, UDAEnableTagReadback false
BEGIN

REGION Network 1: BFT 61 Rework 32
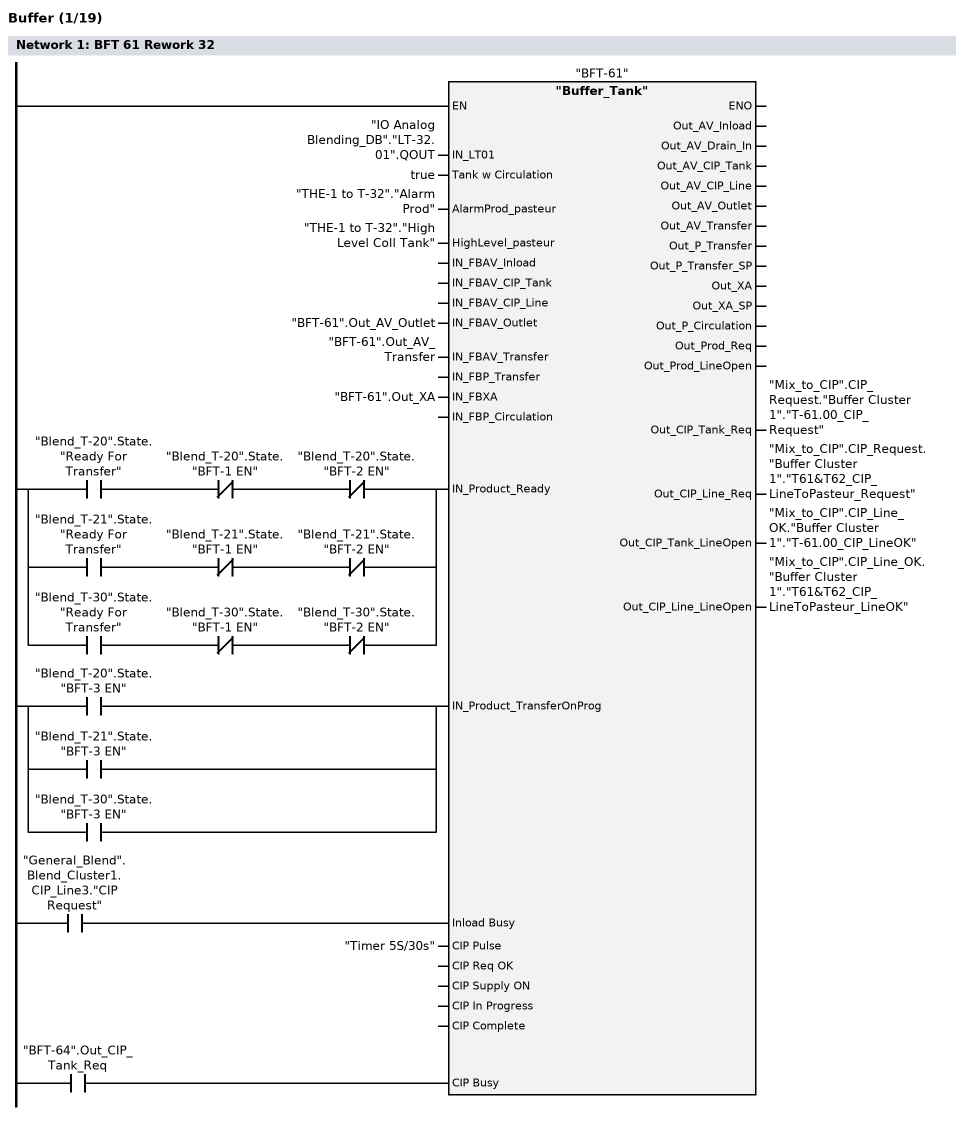
   RUNG wire#powerrail
      "BFT-61"(IN_Product_Ready := wire#w1, IN_Product_TransferOnProg := wire#w2, "Inload Busy" := wire#w3, "CIP Busy" := wire#w4, IN_LT01 := "IO Analog Blending_DB"."LT-32.01".QOUT, "Tank w Circulation" := true, AlarmProd_pasteur := "THE-1 to T-32"."Alarm Prod", HighLevel_pasteur := "THE-1 to T-32"."High Level Coll Tank", IN_FBAV_Inload :=, IN_FBAV_CIP_Tank :=, IN_FBAV_CIP_Line :=, IN_FBAV_Outlet := "BFT-61".Out_AV_Outlet, IN_FBAV_Transfer := "BFT-61".Out_AV_Transfer, IN_FBP_Transfer :=, IN_FBXA := "BFT-61".Out_XA, IN_FBP_Circulation :=, "CIP Pulse" := "Timer 5S/30s", "CIP Req OK" :=, "CIP Supply ON" :=, "CIP In Progress" :=, "CIP Complete" :=, Out_AV_Inload =>, Out_AV_Drain_In =>, Out_AV_CIP_Tank =>, Out_AV_CIP_Line =>, Out_AV_Outlet =>, Out_AV_Transfer =>, Out_P_Transfer =>, Out_P_Transfer_SP =>, Out_XA =>, Out_XA_SP =>, Out_P_Circulation =>, Out_Prod_Req =>, Out_Prod_LineOpen =>, Out_CIP_Tank_Req => "Mix_to_CIP".CIP_Request."Buffer Cluster 1"."T-61.00_CIP_Request", Out_CIP_Line_Req => "Mix_to_CIP".CIP_Request."Buffer Cluster 1"."T61&T62_CIP_LineToPasteur_Request", Out_CIP_Tank_LineOpen => "Mix_to_CIP".CIP_Line_OK."Buffer Cluster 1"."T-61.00_CIP_LineOK", Out_CIP_Line_LineOpen => "Mix_to_CIP".CIP_Line_OK."Buffer Cluster 1"."T61&T62_CIP_LineToPasteur_LineOK")
   END_RUNG
   RUNG wire#powerrail
      Contact( "Blend_T-20".State."Ready For Transfer" )
      I_Contact( "Blend_T-20".State."BFT-1 EN" )
      I_Contact( "Blend_T-20".State."BFT-2 EN" )
   END_RUNG wire#w1
   RUNG wire#powerrail
      Contact( "Blend_T-21".State."Ready For Transfer" )
      I_Contact( "Blend_T-21".State."BFT-1 EN" )
      I_Contact( "Blend_T-21".State."BFT-2 EN" )
   END_RUNG wire#w1
   RUNG wire#powerrail
      Contact( "Blend_T-30".State."Ready For Transfer" )
      I_Contact( "Blend_T-30".State."BFT-1 EN" )
      I_Contact( "Blend_T-30".State."BFT-2 EN" )
   END_RUNG wire#w1
   RUNG wire#powerrail
      Contact( "Blend_T-20".State."BFT-3 EN" )
   END_RUNG wire#w2
   RUNG wire#powerrail
      Contact( "Blend_T-21".State."BFT-3 EN" )
   END_RUNG wire#w2
   RUNG wire#powerrail
      Contact( "Blend_T-30".State."BFT-3 EN" )
   END_RUNG wire#w2
   RUNG wire#powerrail
      Contact( "General_Blend".Blend_Cluster1.CIP_Line3."CIP Request" )
   END_RUNG wire#w3
   RUNG wire#powerrail
      Contact( "BFT-64".Out_CIP_Tank_Req )
   END_RUNG wire#w4
   // the same network as SCL:
   "BFT-61"(IN_LT01 := "IO Analog Blending_DB"."LT-32.01".QOUT,   // "Buffer_Tank"
            "Tank w Circulation" := true,
            AlarmProd_pasteur := "THE-1 to T-32"."Alarm Prod",
            HighLevel_pasteur := "THE-1 to T-32"."High Level Coll Tank",
            IN_FBAV_Outlet := "BFT-61".Out_AV_Outlet,
            IN_FBAV_Transfer := "BFT-61".Out_AV_Transfer,
            IN_FBXA := "BFT-61".Out_XA,
            IN_Product_Ready := ("Blend_T-20".State."Ready For Transfer" AND NOT "Blend_T-20".State."BFT-1 EN" AND NOT "Blend_T-20".State."BFT-2 EN") OR ("Blend_T-21".State."Ready For Transfer" AND NOT "Blend_T-21".State."BFT-1 EN" AND NOT "Blend_T-21".State."BFT-2 EN") OR ("Blend_T-30".State."Ready For Transfer" AND NOT "Blend_T-30".State."BFT-1 EN" AND NOT "Blend_T-30".State."BFT-2 EN"),
            IN_Product_TransferOnProg := "Blend_T-20".State."BFT-3 EN" OR "Blend_T-21".State."BFT-3 EN" OR "Blend_T-30".State."BFT-3 EN",
            "Inload Busy" := "General_Blend".Blend_Cluster1.CIP_Line3."CIP Request",
            "CIP Pulse" := "Timer 5S/30s",
            "CIP Busy" := "BFT-64".Out_CIP_Tank_Req,
            Out_CIP_Tank_Req => "Mix_to_CIP".CIP_Request."Buffer Cluster 1"."T-61.00_CIP_Request",
            Out_CIP_Line_Req => "Mix_to_CIP".CIP_Request."Buffer Cluster 1"."T61&T62_CIP_LineToPasteur_Request",
            Out_CIP_Tank_LineOpen => "Mix_to_CIP".CIP_Line_OK."Buffer Cluster 1"."T-61.00_CIP_LineOK",
            Out_CIP_Line_LineOpen => "Mix_to_CIP".CIP_Line_OK."Buffer Cluster 1"."T61&T62_CIP_LineToPasteur_LineOK");
END_REGION

REGION Network 2: BFT 61 Feedback Instrument
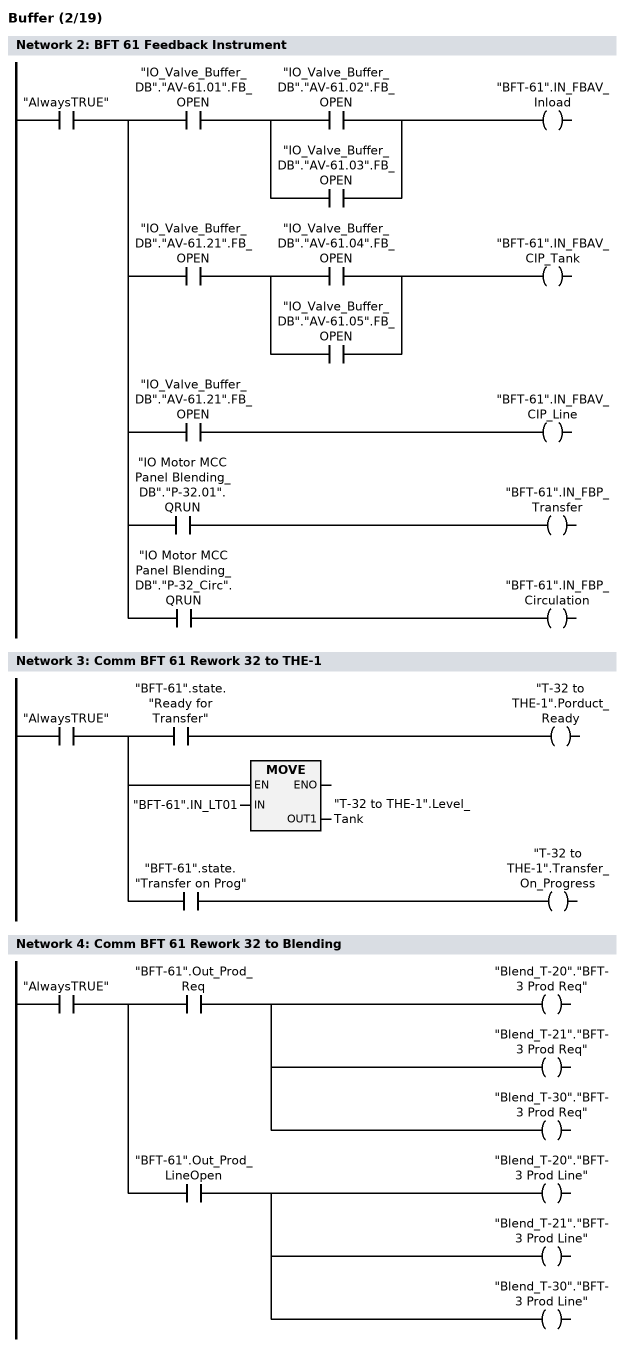
   RUNG wire#powerrail
      Contact( "AlwaysTRUE" )
      wire#w1
      Contact( "IO_Valve_Buffer_DB"."AV-61.01".FB_OPEN )
      wire#w2
      Contact( "IO_Valve_Buffer_DB"."AV-61.02".FB_OPEN )
      wire#w3
      Coil( "BFT-61".IN_FBAV_Inload )
   END_RUNG
   RUNG wire#w2
      Contact( "IO_Valve_Buffer_DB"."AV-61.03".FB_OPEN )
   END_RUNG wire#w3
   RUNG wire#w1
      Contact( "IO_Valve_Buffer_DB"."AV-61.21".FB_OPEN )
      wire#w4
      Contact( "IO_Valve_Buffer_DB"."AV-61.04".FB_OPEN )
      wire#w5
      Coil( "BFT-61".IN_FBAV_CIP_Tank )
   END_RUNG
   RUNG wire#w4
      Contact( "IO_Valve_Buffer_DB"."AV-61.05".FB_OPEN )
   END_RUNG wire#w5
   RUNG wire#w1
      Contact( "IO_Valve_Buffer_DB"."AV-61.21".FB_OPEN )
      Coil( "BFT-61".IN_FBAV_CIP_Line )
   END_RUNG
   RUNG wire#w1
      Contact( "IO Motor MCC Panel Blending_DB"."P-32.01".QRUN )
      Coil( "BFT-61".IN_FBP_Transfer )
   END_RUNG
   RUNG wire#w1
      Contact( "IO Motor MCC Panel Blending_DB"."P-32_Circ".QRUN )
      Coil( "BFT-61".IN_FBP_Circulation )
   END_RUNG
   // the same network as SCL:
   "BFT-61".IN_FBAV_Inload := "AlwaysTRUE" AND "IO_Valve_Buffer_DB"."AV-61.01".FB_OPEN AND ("IO_Valve_Buffer_DB"."AV-61.02".FB_OPEN OR "IO_Valve_Buffer_DB"."AV-61.03".FB_OPEN);
   "BFT-61".IN_FBAV_CIP_Tank := "AlwaysTRUE" AND "IO_Valve_Buffer_DB"."AV-61.21".FB_OPEN AND ("IO_Valve_Buffer_DB"."AV-61.04".FB_OPEN OR "IO_Valve_Buffer_DB"."AV-61.05".FB_OPEN);
   "BFT-61".IN_FBAV_CIP_Line := "AlwaysTRUE" AND "IO_Valve_Buffer_DB"."AV-61.21".FB_OPEN;
   "BFT-61".IN_FBP_Transfer := "AlwaysTRUE" AND "IO Motor MCC Panel Blending_DB"."P-32.01".QRUN;
   "BFT-61".IN_FBP_Circulation := "AlwaysTRUE" AND "IO Motor MCC Panel Blending_DB"."P-32_Circ".QRUN;
END_REGION

REGION Network 3: Comm BFT 61 Rework 32 to THE-1
   RUNG wire#powerrail
      Contact( "AlwaysTRUE" )
      wire#w1
      Contact( "BFT-61".state."Ready for Transfer" )
      Coil( "T-32 to THE-1".Porduct_Ready )
   END_RUNG
   RUNG wire#w1
      Move(in := "BFT-61".IN_LT01, out1 => "T-32 to THE-1".Level_Tank)
   END_RUNG
   RUNG wire#w1
      Contact( "BFT-61".state."Transfer on Prog" )
      Coil( "T-32 to THE-1".Transfer_On_Progress )
   END_RUNG
   // the same network as SCL:
   "T-32 to THE-1".Porduct_Ready := "AlwaysTRUE" AND "BFT-61".state."Ready for Transfer";
   IF "AlwaysTRUE" THEN "T-32 to THE-1".Level_Tank := "BFT-61".IN_LT01; END_IF;
   "T-32 to THE-1".Transfer_On_Progress := "AlwaysTRUE" AND "BFT-61".state."Transfer on Prog";
END_REGION

REGION Network 4: Comm BFT 61 Rework 32 to Blending
   RUNG wire#powerrail
      Contact( "AlwaysTRUE" )
      wire#w1
      Contact( "BFT-61".Out_Prod_Req )
      wire#w2
      Coil( "Blend_T-20"."BFT-3 Prod Req" )
   END_RUNG
   RUNG wire#w2
      Coil( "Blend_T-21"."BFT-3 Prod Req" )
   END_RUNG
   RUNG wire#w2
      Coil( "Blend_T-30"."BFT-3 Prod Req" )
   END_RUNG
   RUNG wire#w1
      Contact( "BFT-61".Out_Prod_LineOpen )
      wire#w3
      Coil( "Blend_T-20"."BFT-3 Prod Line" )
   END_RUNG
   RUNG wire#w3
      Coil( "Blend_T-21"."BFT-3 Prod Line" )
   END_RUNG
   RUNG wire#w3
      Coil( "Blend_T-30"."BFT-3 Prod Line" )
   END_RUNG
   // the same network as SCL:
   "Blend_T-20"."BFT-3 Prod Req" := "AlwaysTRUE" AND "BFT-61".Out_Prod_Req;
   "Blend_T-21"."BFT-3 Prod Req" := "Blend_T-20"."BFT-3 Prod Req";
   "Blend_T-30"."BFT-3 Prod Req" := "Blend_T-20"."BFT-3 Prod Req";
   "Blend_T-20"."BFT-3 Prod Line" := "AlwaysTRUE" AND "BFT-61".Out_Prod_LineOpen;
   "Blend_T-21"."BFT-3 Prod Line" := "Blend_T-20"."BFT-3 Prod Line";
   "Blend_T-30"."BFT-3 Prod Line" := "Blend_T-20"."BFT-3 Prod Line";
END_REGION

REGION Network 6: BFT 64 Rework 22
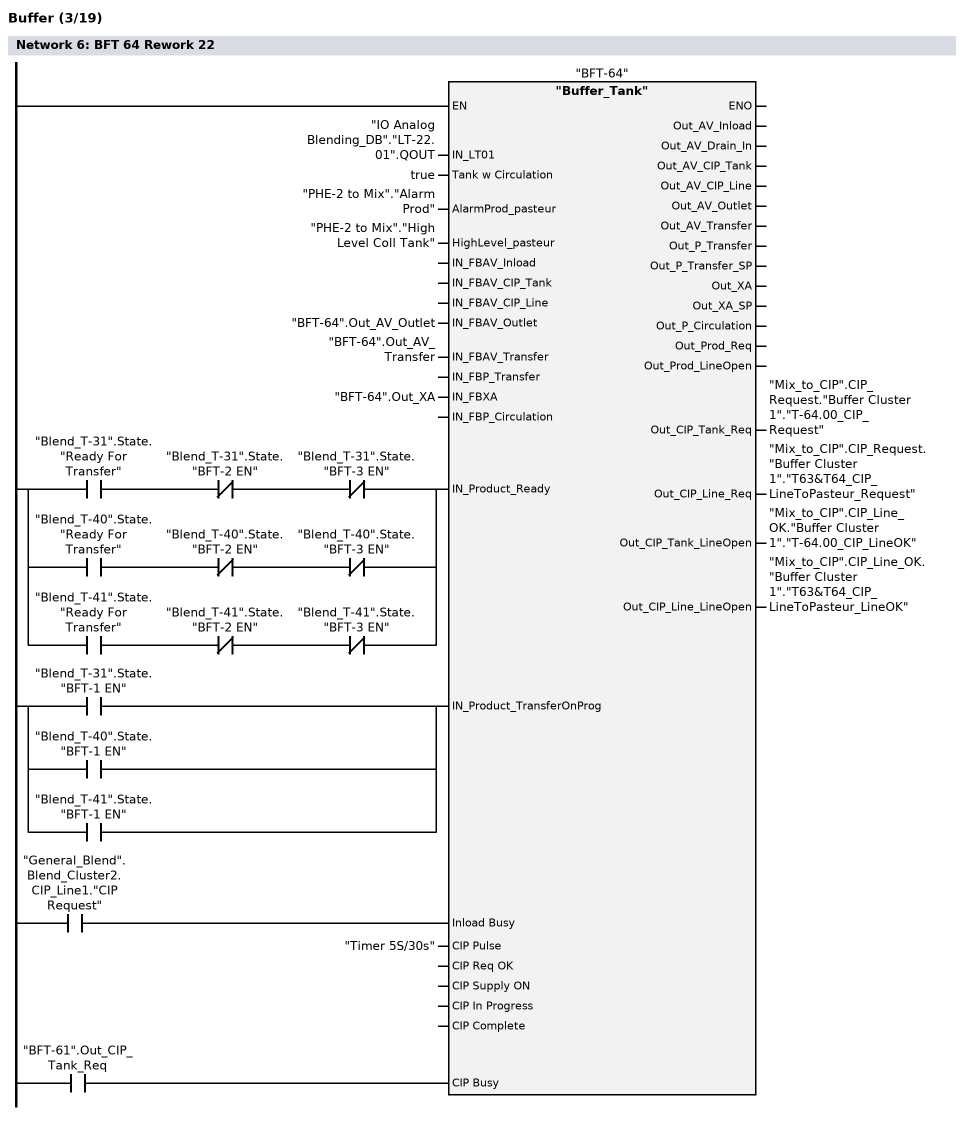
   RUNG wire#powerrail
      "BFT-64"(IN_Product_Ready := wire#w1, IN_Product_TransferOnProg := wire#w2, "Inload Busy" := wire#w3, "CIP Busy" := wire#w4, IN_LT01 := "IO Analog Blending_DB"."LT-22.01".QOUT, "Tank w Circulation" := true, AlarmProd_pasteur := "PHE-2 to Mix"."Alarm Prod", HighLevel_pasteur := "PHE-2 to Mix"."High Level Coll Tank", IN_FBAV_Inload :=, IN_FBAV_CIP_Tank :=, IN_FBAV_CIP_Line :=, IN_FBAV_Outlet := "BFT-64".Out_AV_Outlet, IN_FBAV_Transfer := "BFT-64".Out_AV_Transfer, IN_FBP_Transfer :=, IN_FBXA := "BFT-64".Out_XA, IN_FBP_Circulation :=, "CIP Pulse" := "Timer 5S/30s", "CIP Req OK" :=, "CIP Supply ON" :=, "CIP In Progress" :=, "CIP Complete" :=, Out_AV_Inload =>, Out_AV_Drain_In =>, Out_AV_CIP_Tank =>, Out_AV_CIP_Line =>, Out_AV_Outlet =>, Out_AV_Transfer =>, Out_P_Transfer =>, Out_P_Transfer_SP =>, Out_XA =>, Out_XA_SP =>, Out_P_Circulation =>, Out_Prod_Req =>, Out_Prod_LineOpen =>, Out_CIP_Tank_Req => "Mix_to_CIP".CIP_Request."Buffer Cluster 1"."T-64.00_CIP_Request", Out_CIP_Line_Req => "Mix_to_CIP".CIP_Request."Buffer Cluster 1"."T63&T64_CIP_LineToPasteur_Request", Out_CIP_Tank_LineOpen => "Mix_to_CIP".CIP_Line_OK."Buffer Cluster 1"."T-64.00_CIP_LineOK", Out_CIP_Line_LineOpen => "Mix_to_CIP".CIP_Line_OK."Buffer Cluster 1"."T63&T64_CIP_LineToPasteur_LineOK")
   END_RUNG
   RUNG wire#powerrail
      Contact( "Blend_T-31".State."Ready For Transfer" )
      I_Contact( "Blend_T-31".State."BFT-2 EN" )
      I_Contact( "Blend_T-31".State."BFT-3 EN" )
   END_RUNG wire#w1
   RUNG wire#powerrail
      Contact( "Blend_T-40".State."Ready For Transfer" )
      I_Contact( "Blend_T-40".State."BFT-2 EN" )
      I_Contact( "Blend_T-40".State."BFT-3 EN" )
   END_RUNG wire#w1
   RUNG wire#powerrail
      Contact( "Blend_T-41".State."Ready For Transfer" )
      I_Contact( "Blend_T-41".State."BFT-2 EN" )
      I_Contact( "Blend_T-41".State."BFT-3 EN" )
   END_RUNG wire#w1
   RUNG wire#powerrail
      Contact( "Blend_T-31".State."BFT-1 EN" )
   END_RUNG wire#w2
   RUNG wire#powerrail
      Contact( "Blend_T-40".State."BFT-1 EN" )
   END_RUNG wire#w2
   RUNG wire#powerrail
      Contact( "Blend_T-41".State."BFT-1 EN" )
   END_RUNG wire#w2
   RUNG wire#powerrail
      Contact( "General_Blend".Blend_Cluster2.CIP_Line1."CIP Request" )
   END_RUNG wire#w3
   RUNG wire#powerrail
      Contact( "BFT-61".Out_CIP_Tank_Req )
   END_RUNG wire#w4
   // the same network as SCL:
   "BFT-64"(IN_LT01 := "IO Analog Blending_DB"."LT-22.01".QOUT,   // "Buffer_Tank"
            "Tank w Circulation" := true,
            AlarmProd_pasteur := "PHE-2 to Mix"."Alarm Prod",
            HighLevel_pasteur := "PHE-2 to Mix"."High Level Coll Tank",
            IN_FBAV_Outlet := "BFT-64".Out_AV_Outlet,
            IN_FBAV_Transfer := "BFT-64".Out_AV_Transfer,
            IN_FBXA := "BFT-64".Out_XA,
            IN_Product_Ready := ("Blend_T-31".State."Ready For Transfer" AND NOT "Blend_T-31".State."BFT-2 EN" AND NOT "Blend_T-31".State."BFT-3 EN") OR ("Blend_T-40".State."Ready For Transfer" AND NOT "Blend_T-40".State."BFT-2 EN" AND NOT "Blend_T-40".State."BFT-3 EN") OR ("Blend_T-41".State."Ready For Transfer" AND NOT "Blend_T-41".State."BFT-2 EN" AND NOT "Blend_T-41".State."BFT-3 EN"),
            IN_Product_TransferOnProg := "Blend_T-31".State."BFT-1 EN" OR "Blend_T-40".State."BFT-1 EN" OR "Blend_T-41".State."BFT-1 EN",
            "Inload Busy" := "General_Blend".Blend_Cluster2.CIP_Line1."CIP Request",
            "CIP Pulse" := "Timer 5S/30s",
            "CIP Busy" := "BFT-61".Out_CIP_Tank_Req,
            Out_CIP_Tank_Req => "Mix_to_CIP".CIP_Request."Buffer Cluster 1"."T-64.00_CIP_Request",
            Out_CIP_Line_Req => "Mix_to_CIP".CIP_Request."Buffer Cluster 1"."T63&T64_CIP_LineToPasteur_Request",
            Out_CIP_Tank_LineOpen => "Mix_to_CIP".CIP_Line_OK."Buffer Cluster 1"."T-64.00_CIP_LineOK",
            Out_CIP_Line_LineOpen => "Mix_to_CIP".CIP_Line_OK."Buffer Cluster 1"."T63&T64_CIP_LineToPasteur_LineOK");
END_REGION

REGION Network 7: BFT 64 Feedback Instrument
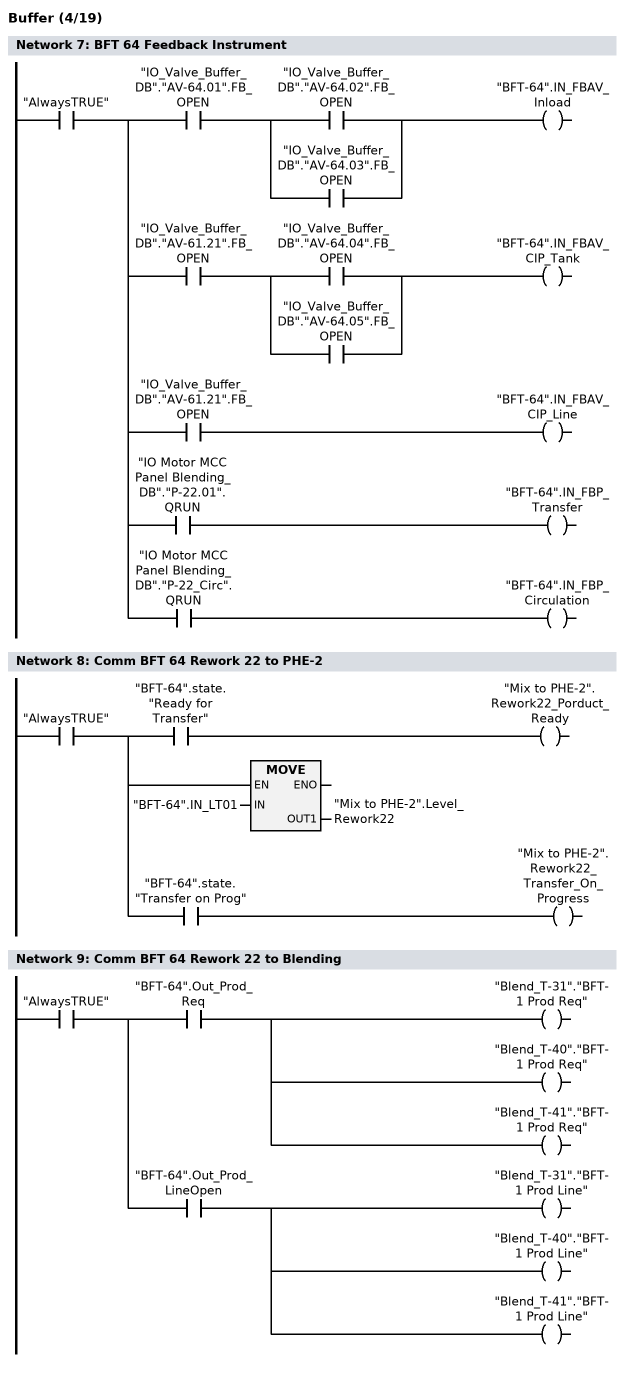
   RUNG wire#powerrail
      Contact( "AlwaysTRUE" )
      wire#w1
      Contact( "IO_Valve_Buffer_DB"."AV-64.01".FB_OPEN )
      wire#w2
      Contact( "IO_Valve_Buffer_DB"."AV-64.02".FB_OPEN )
      wire#w3
      Coil( "BFT-64".IN_FBAV_Inload )
   END_RUNG
   RUNG wire#w2
      Contact( "IO_Valve_Buffer_DB"."AV-64.03".FB_OPEN )
   END_RUNG wire#w3
   RUNG wire#w1
      Contact( "IO_Valve_Buffer_DB"."AV-61.21".FB_OPEN )
      wire#w4
      Contact( "IO_Valve_Buffer_DB"."AV-64.04".FB_OPEN )
      wire#w5
      Coil( "BFT-64".IN_FBAV_CIP_Tank )
   END_RUNG
   RUNG wire#w4
      Contact( "IO_Valve_Buffer_DB"."AV-64.05".FB_OPEN )
   END_RUNG wire#w5
   RUNG wire#w1
      Contact( "IO_Valve_Buffer_DB"."AV-61.21".FB_OPEN )
      Coil( "BFT-64".IN_FBAV_CIP_Line )
   END_RUNG
   RUNG wire#w1
      Contact( "IO Motor MCC Panel Blending_DB"."P-22.01".QRUN )
      Coil( "BFT-64".IN_FBP_Transfer )
   END_RUNG
   RUNG wire#w1
      Contact( "IO Motor MCC Panel Blending_DB"."P-22_Circ".QRUN )
      Coil( "BFT-64".IN_FBP_Circulation )
   END_RUNG
   // the same network as SCL:
   "BFT-64".IN_FBAV_Inload := "AlwaysTRUE" AND "IO_Valve_Buffer_DB"."AV-64.01".FB_OPEN AND ("IO_Valve_Buffer_DB"."AV-64.02".FB_OPEN OR "IO_Valve_Buffer_DB"."AV-64.03".FB_OPEN);
   "BFT-64".IN_FBAV_CIP_Tank := "AlwaysTRUE" AND "IO_Valve_Buffer_DB"."AV-61.21".FB_OPEN AND ("IO_Valve_Buffer_DB"."AV-64.04".FB_OPEN OR "IO_Valve_Buffer_DB"."AV-64.05".FB_OPEN);
   "BFT-64".IN_FBAV_CIP_Line := "AlwaysTRUE" AND "IO_Valve_Buffer_DB"."AV-61.21".FB_OPEN;
   "BFT-64".IN_FBP_Transfer := "AlwaysTRUE" AND "IO Motor MCC Panel Blending_DB"."P-22.01".QRUN;
   "BFT-64".IN_FBP_Circulation := "AlwaysTRUE" AND "IO Motor MCC Panel Blending_DB"."P-22_Circ".QRUN;
END_REGION

REGION Network 8: Comm BFT 64 Rework 22 to PHE-2
   RUNG wire#powerrail
      Contact( "AlwaysTRUE" )
      wire#w1
      Contact( "BFT-64".state."Ready for Transfer" )
      Coil( "Mix to PHE-2".Rework22_Porduct_Ready )
   END_RUNG
   RUNG wire#w1
      Move(in := "BFT-64".IN_LT01, out1 => "Mix to PHE-2".Level_Rework22)
   END_RUNG
   RUNG wire#w1
      Contact( "BFT-64".state."Transfer on Prog" )
      Coil( "Mix to PHE-2".Rework22_Transfer_On_Progress )
   END_RUNG
   // the same network as SCL:
   "Mix to PHE-2".Rework22_Porduct_Ready := "AlwaysTRUE" AND "BFT-64".state."Ready for Transfer";
   IF "AlwaysTRUE" THEN "Mix to PHE-2".Level_Rework22 := "BFT-64".IN_LT01; END_IF;
   "Mix to PHE-2".Rework22_Transfer_On_Progress := "AlwaysTRUE" AND "BFT-64".state."Transfer on Prog";
END_REGION

REGION Network 9: Comm BFT 64 Rework 22 to Blending
   RUNG wire#powerrail
      Contact( "AlwaysTRUE" )
      wire#w1
      Contact( "BFT-64".Out_Prod_Req )
      wire#w2
      Coil( "Blend_T-31"."BFT-1 Prod Req" )
   END_RUNG
   RUNG wire#w2
      Coil( "Blend_T-40"."BFT-1 Prod Req" )
   END_RUNG
   RUNG wire#w2
      Coil( "Blend_T-41"."BFT-1 Prod Req" )
   END_RUNG
   RUNG wire#w1
      Contact( "BFT-64".Out_Prod_LineOpen )
      wire#w3
      Coil( "Blend_T-31"."BFT-1 Prod Line" )
   END_RUNG
   RUNG wire#w3
      Coil( "Blend_T-40"."BFT-1 Prod Line" )
   END_RUNG
   RUNG wire#w3
      Coil( "Blend_T-41"."BFT-1 Prod Line" )
   END_RUNG
   // the same network as SCL:
   "Blend_T-31"."BFT-1 Prod Req" := "AlwaysTRUE" AND "BFT-64".Out_Prod_Req;
   "Blend_T-40"."BFT-1 Prod Req" := "Blend_T-31"."BFT-1 Prod Req";
   "Blend_T-41"."BFT-1 Prod Req" := "Blend_T-31"."BFT-1 Prod Req";
   "Blend_T-31"."BFT-1 Prod Line" := "AlwaysTRUE" AND "BFT-64".Out_Prod_LineOpen;
   "Blend_T-40"."BFT-1 Prod Line" := "Blend_T-31"."BFT-1 Prod Line";
   "Blend_T-41"."BFT-1 Prod Line" := "Blend_T-31"."BFT-1 Prod Line";
END_REGION

REGION Network 11: BFT 65
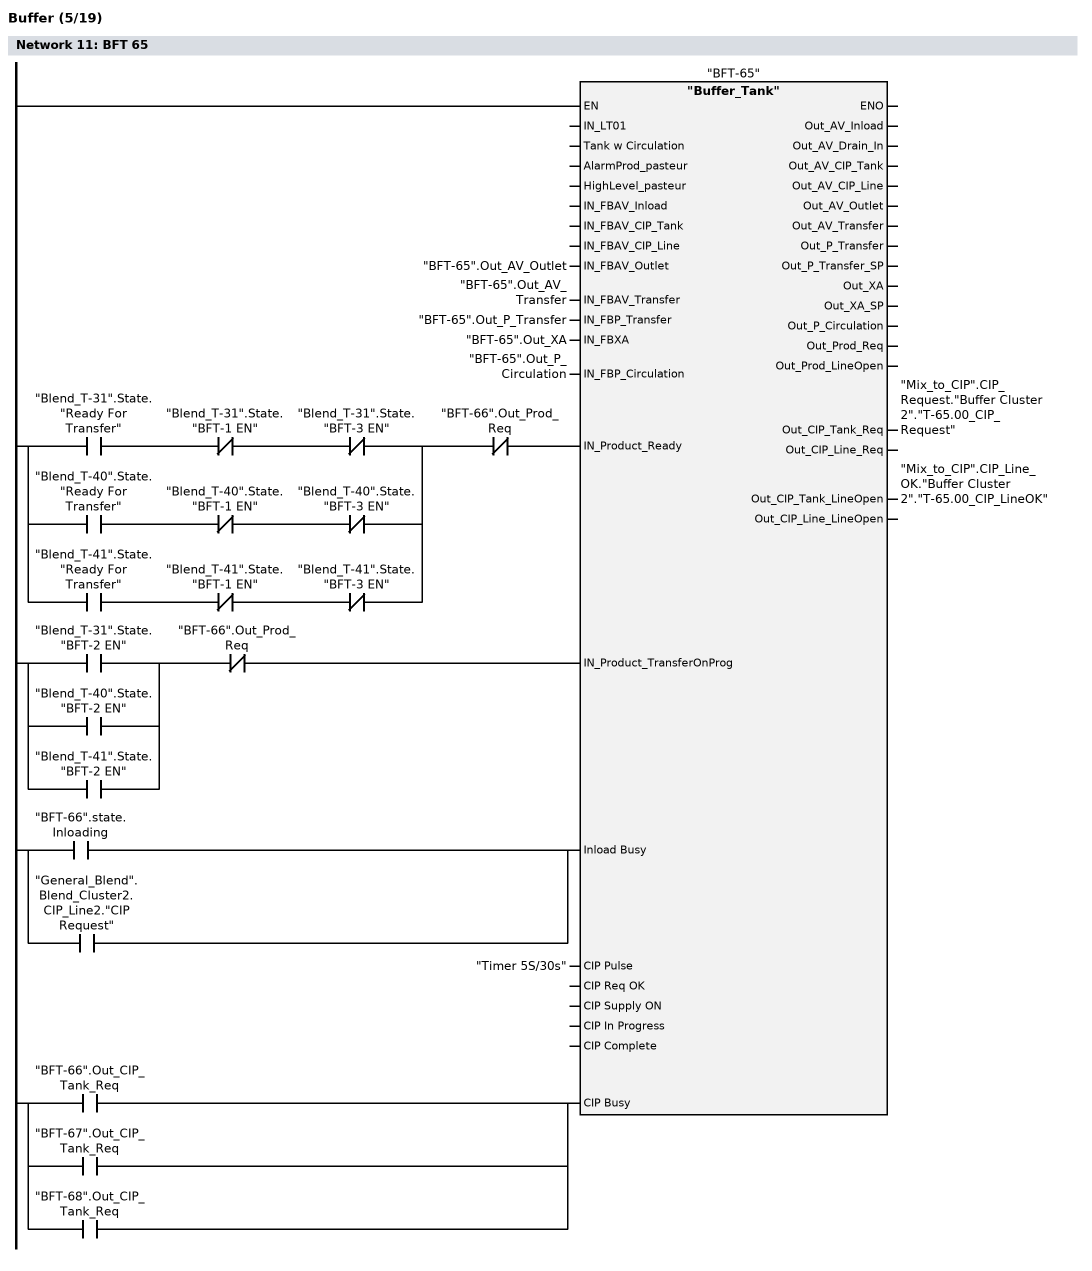
   RUNG wire#powerrail
      "BFT-65"(IN_Product_Ready := wire#w2, IN_Product_TransferOnProg := wire#w4, "Inload Busy" := wire#w5, "CIP Busy" := wire#w6, IN_LT01 :=, "Tank w Circulation" :=, AlarmProd_pasteur :=, HighLevel_pasteur :=, IN_FBAV_Inload :=, IN_FBAV_CIP_Tank :=, IN_FBAV_CIP_Line :=, IN_FBAV_Outlet := "BFT-65".Out_AV_Outlet, IN_FBAV_Transfer := "BFT-65".Out_AV_Transfer, IN_FBP_Transfer := "BFT-65".Out_P_Transfer, IN_FBXA := "BFT-65".Out_XA, IN_FBP_Circulation := "BFT-65".Out_P_Circulation, "CIP Pulse" := "Timer 5S/30s", "CIP Req OK" :=, "CIP Supply ON" :=, "CIP In Progress" :=, "CIP Complete" :=, Out_AV_Inload =>, Out_AV_Drain_In =>, Out_AV_CIP_Tank =>, Out_AV_CIP_Line =>, Out_AV_Outlet =>, Out_AV_Transfer =>, Out_P_Transfer =>, Out_P_Transfer_SP =>, Out_XA =>, Out_XA_SP =>, Out_P_Circulation =>, Out_Prod_Req =>, Out_Prod_LineOpen =>, Out_CIP_Tank_Req => "Mix_to_CIP".CIP_Request."Buffer Cluster 2"."T-65.00_CIP_Request", Out_CIP_Line_Req =>, Out_CIP_Tank_LineOpen => "Mix_to_CIP".CIP_Line_OK."Buffer Cluster 2"."T-65.00_CIP_LineOK", Out_CIP_Line_LineOpen =>)
   END_RUNG
   RUNG wire#powerrail
      Contact( "Blend_T-31".State."Ready For Transfer" )
      I_Contact( "Blend_T-31".State."BFT-1 EN" )
      I_Contact( "Blend_T-31".State."BFT-3 EN" )
      wire#w1
      I_Contact( "BFT-66".Out_Prod_Req )
   END_RUNG wire#w2
   RUNG wire#powerrail
      Contact( "Blend_T-40".State."Ready For Transfer" )
      I_Contact( "Blend_T-40".State."BFT-1 EN" )
      I_Contact( "Blend_T-40".State."BFT-3 EN" )
   END_RUNG wire#w1
   RUNG wire#powerrail
      Contact( "Blend_T-41".State."Ready For Transfer" )
      I_Contact( "Blend_T-41".State."BFT-1 EN" )
      I_Contact( "Blend_T-41".State."BFT-3 EN" )
   END_RUNG wire#w1
   RUNG wire#powerrail
      Contact( "Blend_T-31".State."BFT-2 EN" )
      wire#w3
      I_Contact( "BFT-66".Out_Prod_Req )
   END_RUNG wire#w4
   RUNG wire#powerrail
      Contact( "Blend_T-40".State."BFT-2 EN" )
   END_RUNG wire#w3
   RUNG wire#powerrail
      Contact( "Blend_T-41".State."BFT-2 EN" )
   END_RUNG wire#w3
   RUNG wire#powerrail
      Contact( "BFT-66".state.Inloading )
   END_RUNG wire#w5
   RUNG wire#powerrail
      Contact( "General_Blend".Blend_Cluster2.CIP_Line2."CIP Request" )
   END_RUNG wire#w5
   RUNG wire#powerrail
      Contact( "BFT-66".Out_CIP_Tank_Req )
   END_RUNG wire#w6
   RUNG wire#powerrail
      Contact( "BFT-67".Out_CIP_Tank_Req )
   END_RUNG wire#w6
   RUNG wire#powerrail
      Contact( "BFT-68".Out_CIP_Tank_Req )
   END_RUNG wire#w6
   // the same network as SCL:
   "BFT-65"(IN_FBAV_Outlet := "BFT-65".Out_AV_Outlet,   // "Buffer_Tank"
            IN_FBAV_Transfer := "BFT-65".Out_AV_Transfer,
            IN_FBP_Transfer := "BFT-65".Out_P_Transfer,
            IN_FBXA := "BFT-65".Out_XA,
            IN_FBP_Circulation := "BFT-65".Out_P_Circulation,
            IN_Product_Ready := (("Blend_T-31".State."Ready For Transfer" AND NOT "Blend_T-31".State."BFT-1 EN" AND NOT "Blend_T-31".State."BFT-3 EN") OR ("Blend_T-40".State."Ready For Transfer" AND NOT "Blend_T-40".State."BFT-1 EN" AND NOT "Blend_T-40".State."BFT-3 EN") OR ("Blend_T-41".State."Ready For Transfer" AND NOT "Blend_T-41".State."BFT-1 EN" AND NOT "Blend_T-41".State."BFT-3 EN")) AND NOT "BFT-66".Out_Prod_Req,
            IN_Product_TransferOnProg := ("Blend_T-31".State."BFT-2 EN" OR "Blend_T-40".State."BFT-2 EN" OR "Blend_T-41".State."BFT-2 EN") AND NOT "BFT-66".Out_Prod_Req,
            "Inload Busy" := "BFT-66".state.Inloading OR "General_Blend".Blend_Cluster2.CIP_Line2."CIP Request",
            "CIP Pulse" := "Timer 5S/30s",
            "CIP Busy" := "BFT-66".Out_CIP_Tank_Req OR "BFT-67".Out_CIP_Tank_Req OR "BFT-68".Out_CIP_Tank_Req,
            Out_CIP_Tank_Req => "Mix_to_CIP".CIP_Request."Buffer Cluster 2"."T-65.00_CIP_Request",
            Out_CIP_Tank_LineOpen => "Mix_to_CIP".CIP_Line_OK."Buffer Cluster 2"."T-65.00_CIP_LineOK");
END_REGION

REGION Network 12: BFT 65 Feedback Instrument
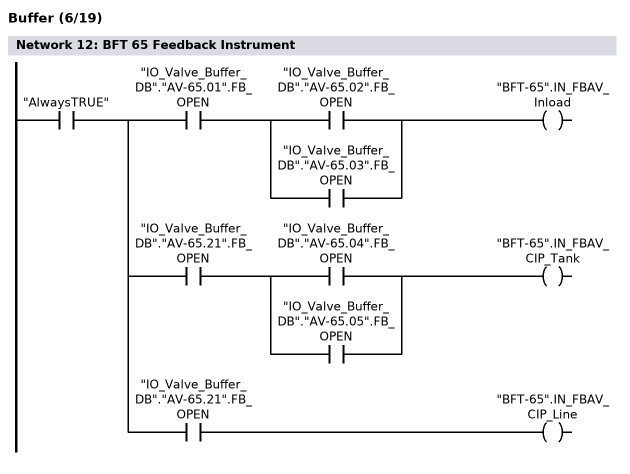
   RUNG wire#powerrail
      Contact( "AlwaysTRUE" )
      wire#w1
      Contact( "IO_Valve_Buffer_DB"."AV-65.01".FB_OPEN )
      wire#w2
      Contact( "IO_Valve_Buffer_DB"."AV-65.02".FB_OPEN )
      wire#w3
      Coil( "BFT-65".IN_FBAV_Inload )
   END_RUNG
   RUNG wire#w2
      Contact( "IO_Valve_Buffer_DB"."AV-65.03".FB_OPEN )
   END_RUNG wire#w3
   RUNG wire#w1
      Contact( "IO_Valve_Buffer_DB"."AV-65.21".FB_OPEN )
      wire#w4
      Contact( "IO_Valve_Buffer_DB"."AV-65.04".FB_OPEN )
      wire#w5
      Coil( "BFT-65".IN_FBAV_CIP_Tank )
   END_RUNG
   RUNG wire#w4
      Contact( "IO_Valve_Buffer_DB"."AV-65.05".FB_OPEN )
   END_RUNG wire#w5
   RUNG wire#w1
      Contact( "IO_Valve_Buffer_DB"."AV-65.21".FB_OPEN )
      Coil( "BFT-65".IN_FBAV_CIP_Line )
   END_RUNG
   // the same network as SCL:
   "BFT-65".IN_FBAV_Inload := "AlwaysTRUE" AND "IO_Valve_Buffer_DB"."AV-65.01".FB_OPEN AND ("IO_Valve_Buffer_DB"."AV-65.02".FB_OPEN OR "IO_Valve_Buffer_DB"."AV-65.03".FB_OPEN);
   "BFT-65".IN_FBAV_CIP_Tank := "AlwaysTRUE" AND "IO_Valve_Buffer_DB"."AV-65.21".FB_OPEN AND ("IO_Valve_Buffer_DB"."AV-65.04".FB_OPEN OR "IO_Valve_Buffer_DB"."AV-65.05".FB_OPEN);
   "BFT-65".IN_FBAV_CIP_Line := "AlwaysTRUE" AND "IO_Valve_Buffer_DB"."AV-65.21".FB_OPEN;
END_REGION

REGION Network 13: BFT 66
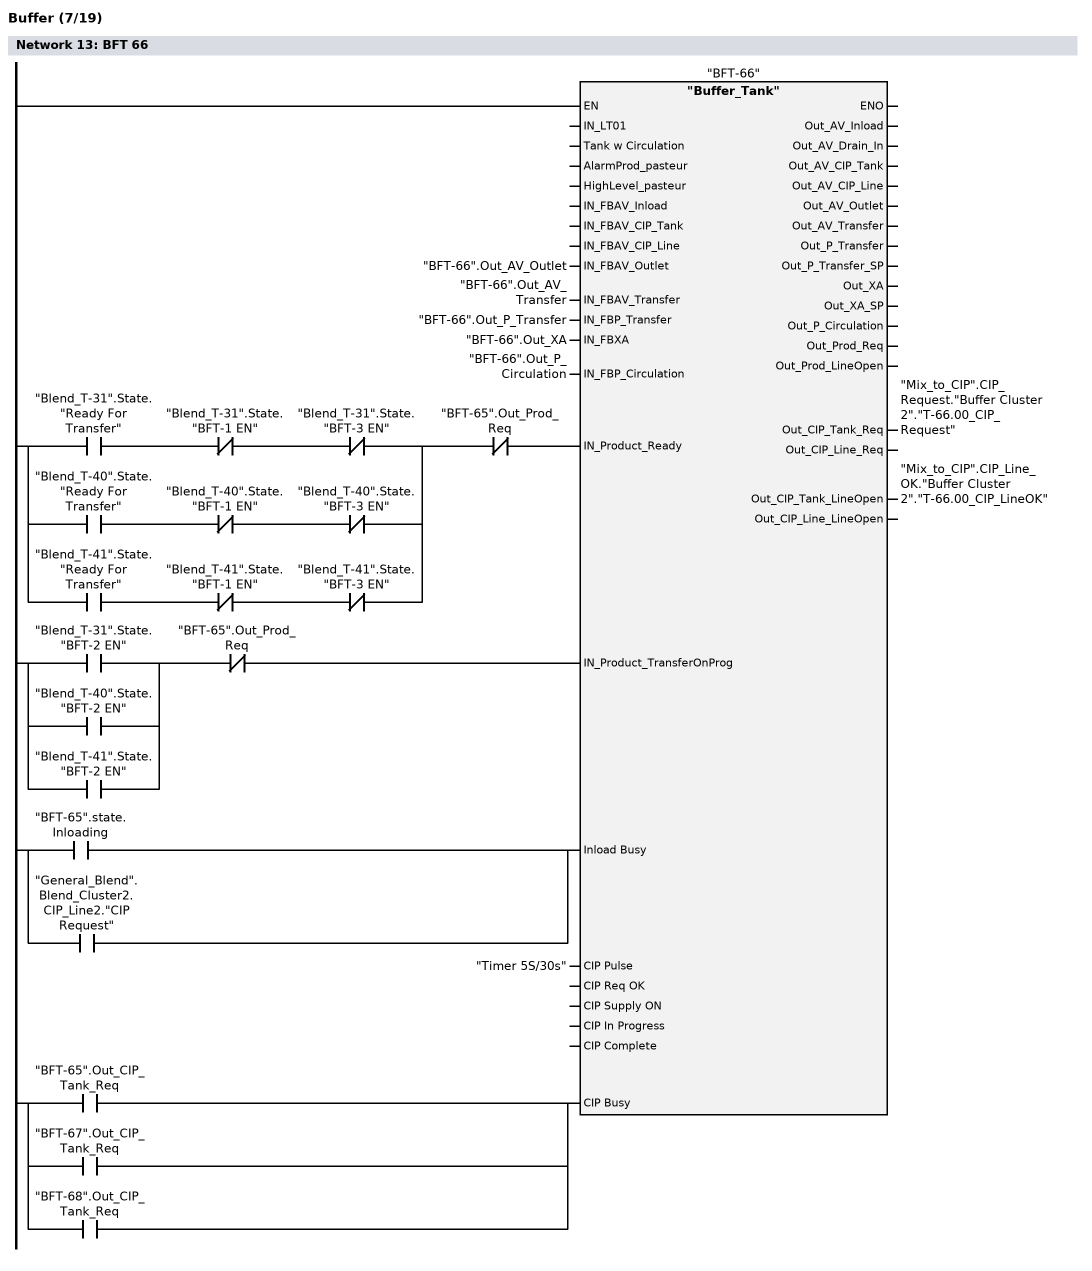
   RUNG wire#powerrail
      "BFT-66"(IN_Product_Ready := wire#w2, IN_Product_TransferOnProg := wire#w4, "Inload Busy" := wire#w5, "CIP Busy" := wire#w6, IN_LT01 :=, "Tank w Circulation" :=, AlarmProd_pasteur :=, HighLevel_pasteur :=, IN_FBAV_Inload :=, IN_FBAV_CIP_Tank :=, IN_FBAV_CIP_Line :=, IN_FBAV_Outlet := "BFT-66".Out_AV_Outlet, IN_FBAV_Transfer := "BFT-66".Out_AV_Transfer, IN_FBP_Transfer := "BFT-66".Out_P_Transfer, IN_FBXA := "BFT-66".Out_XA, IN_FBP_Circulation := "BFT-66".Out_P_Circulation, "CIP Pulse" := "Timer 5S/30s", "CIP Req OK" :=, "CIP Supply ON" :=, "CIP In Progress" :=, "CIP Complete" :=, Out_AV_Inload =>, Out_AV_Drain_In =>, Out_AV_CIP_Tank =>, Out_AV_CIP_Line =>, Out_AV_Outlet =>, Out_AV_Transfer =>, Out_P_Transfer =>, Out_P_Transfer_SP =>, Out_XA =>, Out_XA_SP =>, Out_P_Circulation =>, Out_Prod_Req =>, Out_Prod_LineOpen =>, Out_CIP_Tank_Req => "Mix_to_CIP".CIP_Request."Buffer Cluster 2"."T-66.00_CIP_Request", Out_CIP_Line_Req =>, Out_CIP_Tank_LineOpen => "Mix_to_CIP".CIP_Line_OK."Buffer Cluster 2"."T-66.00_CIP_LineOK", Out_CIP_Line_LineOpen =>)
   END_RUNG
   RUNG wire#powerrail
      Contact( "Blend_T-31".State."Ready For Transfer" )
      I_Contact( "Blend_T-31".State."BFT-1 EN" )
      I_Contact( "Blend_T-31".State."BFT-3 EN" )
      wire#w1
      I_Contact( "BFT-65".Out_Prod_Req )
   END_RUNG wire#w2
   RUNG wire#powerrail
      Contact( "Blend_T-40".State."Ready For Transfer" )
      I_Contact( "Blend_T-40".State."BFT-1 EN" )
      I_Contact( "Blend_T-40".State."BFT-3 EN" )
   END_RUNG wire#w1
   RUNG wire#powerrail
      Contact( "Blend_T-41".State."Ready For Transfer" )
      I_Contact( "Blend_T-41".State."BFT-1 EN" )
      I_Contact( "Blend_T-41".State."BFT-3 EN" )
   END_RUNG wire#w1
   RUNG wire#powerrail
      Contact( "Blend_T-31".State."BFT-2 EN" )
      wire#w3
      I_Contact( "BFT-65".Out_Prod_Req )
   END_RUNG wire#w4
   RUNG wire#powerrail
      Contact( "Blend_T-40".State."BFT-2 EN" )
   END_RUNG wire#w3
   RUNG wire#powerrail
      Contact( "Blend_T-41".State."BFT-2 EN" )
   END_RUNG wire#w3
   RUNG wire#powerrail
      Contact( "BFT-65".state.Inloading )
   END_RUNG wire#w5
   RUNG wire#powerrail
      Contact( "General_Blend".Blend_Cluster2.CIP_Line2."CIP Request" )
   END_RUNG wire#w5
   RUNG wire#powerrail
      Contact( "BFT-65".Out_CIP_Tank_Req )
   END_RUNG wire#w6
   RUNG wire#powerrail
      Contact( "BFT-67".Out_CIP_Tank_Req )
   END_RUNG wire#w6
   RUNG wire#powerrail
      Contact( "BFT-68".Out_CIP_Tank_Req )
   END_RUNG wire#w6
   // the same network as SCL:
   "BFT-66"(IN_FBAV_Outlet := "BFT-66".Out_AV_Outlet,   // "Buffer_Tank"
            IN_FBAV_Transfer := "BFT-66".Out_AV_Transfer,
            IN_FBP_Transfer := "BFT-66".Out_P_Transfer,
            IN_FBXA := "BFT-66".Out_XA,
            IN_FBP_Circulation := "BFT-66".Out_P_Circulation,
            IN_Product_Ready := (("Blend_T-31".State."Ready For Transfer" AND NOT "Blend_T-31".State."BFT-1 EN" AND NOT "Blend_T-31".State."BFT-3 EN") OR ("Blend_T-40".State."Ready For Transfer" AND NOT "Blend_T-40".State."BFT-1 EN" AND NOT "Blend_T-40".State."BFT-3 EN") OR ("Blend_T-41".State."Ready For Transfer" AND NOT "Blend_T-41".State."BFT-1 EN" AND NOT "Blend_T-41".State."BFT-3 EN")) AND NOT "BFT-65".Out_Prod_Req,
            IN_Product_TransferOnProg := ("Blend_T-31".State."BFT-2 EN" OR "Blend_T-40".State."BFT-2 EN" OR "Blend_T-41".State."BFT-2 EN") AND NOT "BFT-65".Out_Prod_Req,
            "Inload Busy" := "BFT-65".state.Inloading OR "General_Blend".Blend_Cluster2.CIP_Line2."CIP Request",
            "CIP Pulse" := "Timer 5S/30s",
            "CIP Busy" := "BFT-65".Out_CIP_Tank_Req OR "BFT-67".Out_CIP_Tank_Req OR "BFT-68".Out_CIP_Tank_Req,
            Out_CIP_Tank_Req => "Mix_to_CIP".CIP_Request."Buffer Cluster 2"."T-66.00_CIP_Request",
            Out_CIP_Tank_LineOpen => "Mix_to_CIP".CIP_Line_OK."Buffer Cluster 2"."T-66.00_CIP_LineOK");
END_REGION

REGION Network 14: BFT 66 Feedback Instrument
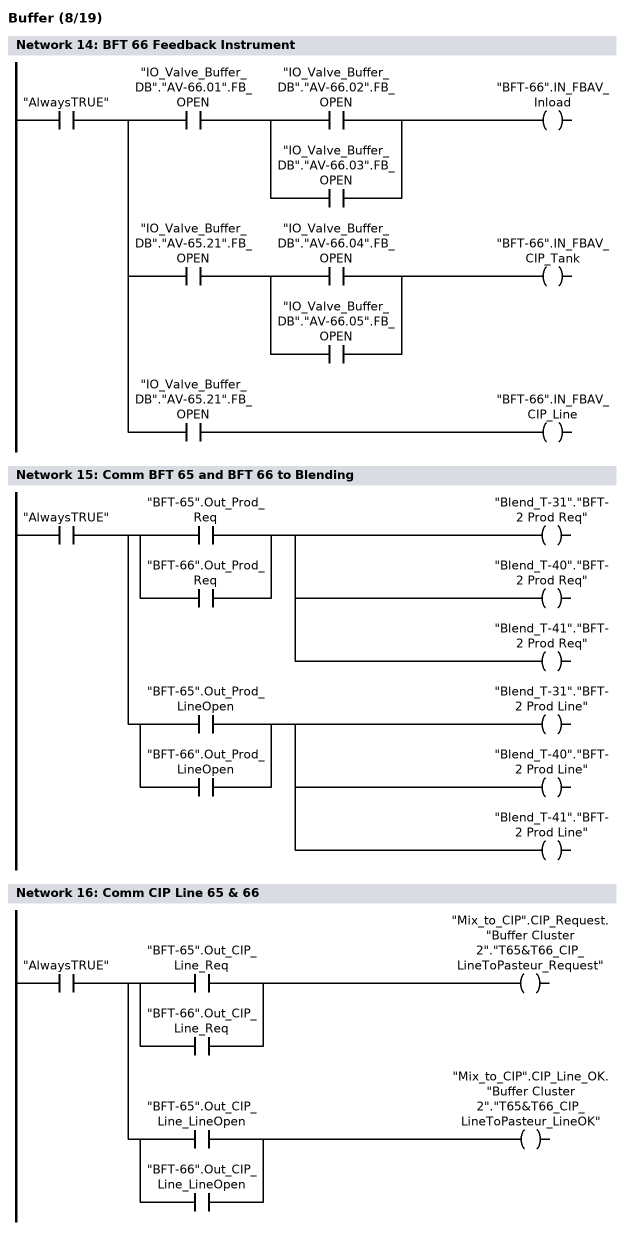
   RUNG wire#powerrail
      Contact( "AlwaysTRUE" )
      wire#w1
      Contact( "IO_Valve_Buffer_DB"."AV-66.01".FB_OPEN )
      wire#w2
      Contact( "IO_Valve_Buffer_DB"."AV-66.02".FB_OPEN )
      wire#w3
      Coil( "BFT-66".IN_FBAV_Inload )
   END_RUNG
   RUNG wire#w2
      Contact( "IO_Valve_Buffer_DB"."AV-66.03".FB_OPEN )
   END_RUNG wire#w3
   RUNG wire#w1
      Contact( "IO_Valve_Buffer_DB"."AV-65.21".FB_OPEN )
      wire#w4
      Contact( "IO_Valve_Buffer_DB"."AV-66.04".FB_OPEN )
      wire#w5
      Coil( "BFT-66".IN_FBAV_CIP_Tank )
   END_RUNG
   RUNG wire#w4
      Contact( "IO_Valve_Buffer_DB"."AV-66.05".FB_OPEN )
   END_RUNG wire#w5
   RUNG wire#w1
      Contact( "IO_Valve_Buffer_DB"."AV-65.21".FB_OPEN )
      Coil( "BFT-66".IN_FBAV_CIP_Line )
   END_RUNG
   // the same network as SCL:
   "BFT-66".IN_FBAV_Inload := "AlwaysTRUE" AND "IO_Valve_Buffer_DB"."AV-66.01".FB_OPEN AND ("IO_Valve_Buffer_DB"."AV-66.02".FB_OPEN OR "IO_Valve_Buffer_DB"."AV-66.03".FB_OPEN);
   "BFT-66".IN_FBAV_CIP_Tank := "AlwaysTRUE" AND "IO_Valve_Buffer_DB"."AV-65.21".FB_OPEN AND ("IO_Valve_Buffer_DB"."AV-66.04".FB_OPEN OR "IO_Valve_Buffer_DB"."AV-66.05".FB_OPEN);
   "BFT-66".IN_FBAV_CIP_Line := "AlwaysTRUE" AND "IO_Valve_Buffer_DB"."AV-65.21".FB_OPEN;
END_REGION

REGION Network 15: Comm BFT 65 and BFT 66 to Blending
   RUNG wire#powerrail
      Contact( "AlwaysTRUE" )
      wire#w1
      Contact( "BFT-65".Out_Prod_Req )
      wire#w2
      Coil( "Blend_T-31"."BFT-2 Prod Req" )
   END_RUNG
   RUNG wire#w1
      Contact( "BFT-66".Out_Prod_Req )
   END_RUNG wire#w2
   RUNG wire#w2
      Coil( "Blend_T-40"."BFT-2 Prod Req" )
   END_RUNG
   RUNG wire#w2
      Coil( "Blend_T-41"."BFT-2 Prod Req" )
   END_RUNG
   RUNG wire#w1
      Contact( "BFT-65".Out_Prod_LineOpen )
      wire#w3
      Coil( "Blend_T-31"."BFT-2 Prod Line" )
   END_RUNG
   RUNG wire#w1
      Contact( "BFT-66".Out_Prod_LineOpen )
   END_RUNG wire#w3
   RUNG wire#w3
      Coil( "Blend_T-40"."BFT-2 Prod Line" )
   END_RUNG
   RUNG wire#w3
      Coil( "Blend_T-41"."BFT-2 Prod Line" )
   END_RUNG
   // the same network as SCL:
   "Blend_T-31"."BFT-2 Prod Req" := "AlwaysTRUE" AND ("BFT-65".Out_Prod_Req OR "BFT-66".Out_Prod_Req);
   "Blend_T-40"."BFT-2 Prod Req" := "Blend_T-31"."BFT-2 Prod Req";
   "Blend_T-41"."BFT-2 Prod Req" := "Blend_T-31"."BFT-2 Prod Req";
   "Blend_T-31"."BFT-2 Prod Line" := "AlwaysTRUE" AND ("BFT-65".Out_Prod_LineOpen OR "BFT-66".Out_Prod_LineOpen);
   "Blend_T-40"."BFT-2 Prod Line" := "Blend_T-31"."BFT-2 Prod Line";
   "Blend_T-41"."BFT-2 Prod Line" := "Blend_T-31"."BFT-2 Prod Line";
END_REGION

REGION Network 16: Comm CIP Line 65 & 66
   RUNG wire#powerrail
      Contact( "AlwaysTRUE" )
      wire#w1
      Contact( "BFT-65".Out_CIP_Line_Req )
      wire#w2
      Coil( "Mix_to_CIP".CIP_Request."Buffer Cluster 2"."T65&T66_CIP_LineToPasteur_Request" )
   END_RUNG
   RUNG wire#w1
      Contact( "BFT-66".Out_CIP_Line_Req )
   END_RUNG wire#w2
   RUNG wire#w1
      Contact( "BFT-65".Out_CIP_Line_LineOpen )
      wire#w3
      Coil( "Mix_to_CIP".CIP_Line_OK."Buffer Cluster 2"."T65&T66_CIP_LineToPasteur_LineOK" )
   END_RUNG
   RUNG wire#w1
      Contact( "BFT-66".Out_CIP_Line_LineOpen )
   END_RUNG wire#w3
   // the same network as SCL:
   "Mix_to_CIP".CIP_Request."Buffer Cluster 2"."T65&T66_CIP_LineToPasteur_Request" := "AlwaysTRUE" AND ("BFT-65".Out_CIP_Line_Req OR "BFT-66".Out_CIP_Line_Req);
   "Mix_to_CIP".CIP_Line_OK."Buffer Cluster 2"."T65&T66_CIP_LineToPasteur_LineOK" := "AlwaysTRUE" AND ("BFT-65".Out_CIP_Line_LineOpen OR "BFT-66".Out_CIP_Line_LineOpen);
END_REGION

REGION Network 18: BFT 67
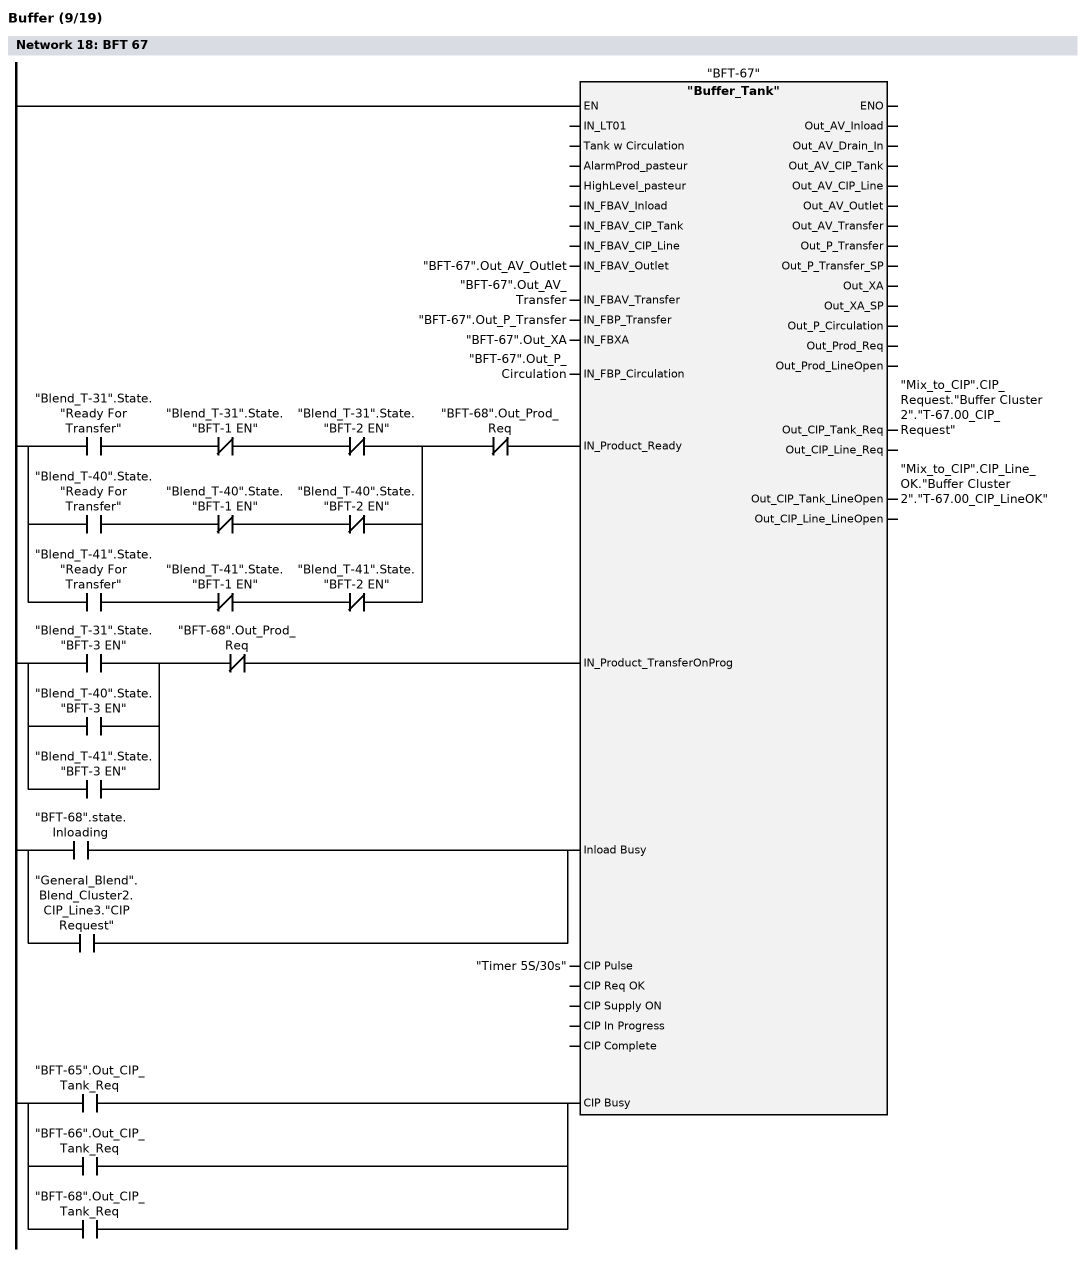
   RUNG wire#powerrail
      "BFT-67"(IN_Product_Ready := wire#w2, IN_Product_TransferOnProg := wire#w4, "Inload Busy" := wire#w5, "CIP Busy" := wire#w6, IN_LT01 :=, "Tank w Circulation" :=, AlarmProd_pasteur :=, HighLevel_pasteur :=, IN_FBAV_Inload :=, IN_FBAV_CIP_Tank :=, IN_FBAV_CIP_Line :=, IN_FBAV_Outlet := "BFT-67".Out_AV_Outlet, IN_FBAV_Transfer := "BFT-67".Out_AV_Transfer, IN_FBP_Transfer := "BFT-67".Out_P_Transfer, IN_FBXA := "BFT-67".Out_XA, IN_FBP_Circulation := "BFT-67".Out_P_Circulation, "CIP Pulse" := "Timer 5S/30s", "CIP Req OK" :=, "CIP Supply ON" :=, "CIP In Progress" :=, "CIP Complete" :=, Out_AV_Inload =>, Out_AV_Drain_In =>, Out_AV_CIP_Tank =>, Out_AV_CIP_Line =>, Out_AV_Outlet =>, Out_AV_Transfer =>, Out_P_Transfer =>, Out_P_Transfer_SP =>, Out_XA =>, Out_XA_SP =>, Out_P_Circulation =>, Out_Prod_Req =>, Out_Prod_LineOpen =>, Out_CIP_Tank_Req => "Mix_to_CIP".CIP_Request."Buffer Cluster 2"."T-67.00_CIP_Request", Out_CIP_Line_Req =>, Out_CIP_Tank_LineOpen => "Mix_to_CIP".CIP_Line_OK."Buffer Cluster 2"."T-67.00_CIP_LineOK", Out_CIP_Line_LineOpen =>)
   END_RUNG
   RUNG wire#powerrail
      Contact( "Blend_T-31".State."Ready For Transfer" )
      I_Contact( "Blend_T-31".State."BFT-1 EN" )
      I_Contact( "Blend_T-31".State."BFT-2 EN" )
      wire#w1
      I_Contact( "BFT-68".Out_Prod_Req )
   END_RUNG wire#w2
   RUNG wire#powerrail
      Contact( "Blend_T-40".State."Ready For Transfer" )
      I_Contact( "Blend_T-40".State."BFT-1 EN" )
      I_Contact( "Blend_T-40".State."BFT-2 EN" )
   END_RUNG wire#w1
   RUNG wire#powerrail
      Contact( "Blend_T-41".State."Ready For Transfer" )
      I_Contact( "Blend_T-41".State."BFT-1 EN" )
      I_Contact( "Blend_T-41".State."BFT-2 EN" )
   END_RUNG wire#w1
   RUNG wire#powerrail
      Contact( "Blend_T-31".State."BFT-3 EN" )
      wire#w3
      I_Contact( "BFT-68".Out_Prod_Req )
   END_RUNG wire#w4
   RUNG wire#powerrail
      Contact( "Blend_T-40".State."BFT-3 EN" )
   END_RUNG wire#w3
   RUNG wire#powerrail
      Contact( "Blend_T-41".State."BFT-3 EN" )
   END_RUNG wire#w3
   RUNG wire#powerrail
      Contact( "BFT-68".state.Inloading )
   END_RUNG wire#w5
   RUNG wire#powerrail
      Contact( "General_Blend".Blend_Cluster2.CIP_Line3."CIP Request" )
   END_RUNG wire#w5
   RUNG wire#powerrail
      Contact( "BFT-65".Out_CIP_Tank_Req )
   END_RUNG wire#w6
   RUNG wire#powerrail
      Contact( "BFT-66".Out_CIP_Tank_Req )
   END_RUNG wire#w6
   RUNG wire#powerrail
      Contact( "BFT-68".Out_CIP_Tank_Req )
   END_RUNG wire#w6
   // the same network as SCL:
   "BFT-67"(IN_FBAV_Outlet := "BFT-67".Out_AV_Outlet,   // "Buffer_Tank"
            IN_FBAV_Transfer := "BFT-67".Out_AV_Transfer,
            IN_FBP_Transfer := "BFT-67".Out_P_Transfer,
            IN_FBXA := "BFT-67".Out_XA,
            IN_FBP_Circulation := "BFT-67".Out_P_Circulation,
            IN_Product_Ready := (("Blend_T-31".State."Ready For Transfer" AND NOT "Blend_T-31".State."BFT-1 EN" AND NOT "Blend_T-31".State."BFT-2 EN") OR ("Blend_T-40".State."Ready For Transfer" AND NOT "Blend_T-40".State."BFT-1 EN" AND NOT "Blend_T-40".State."BFT-2 EN") OR ("Blend_T-41".State."Ready For Transfer" AND NOT "Blend_T-41".State."BFT-1 EN" AND NOT "Blend_T-41".State."BFT-2 EN")) AND NOT "BFT-68".Out_Prod_Req,
            IN_Product_TransferOnProg := ("Blend_T-31".State."BFT-3 EN" OR "Blend_T-40".State."BFT-3 EN" OR "Blend_T-41".State."BFT-3 EN") AND NOT "BFT-68".Out_Prod_Req,
            "Inload Busy" := "BFT-68".state.Inloading OR "General_Blend".Blend_Cluster2.CIP_Line3."CIP Request",
            "CIP Pulse" := "Timer 5S/30s",
            "CIP Busy" := "BFT-65".Out_CIP_Tank_Req OR "BFT-66".Out_CIP_Tank_Req OR "BFT-68".Out_CIP_Tank_Req,
            Out_CIP_Tank_Req => "Mix_to_CIP".CIP_Request."Buffer Cluster 2"."T-67.00_CIP_Request",
            Out_CIP_Tank_LineOpen => "Mix_to_CIP".CIP_Line_OK."Buffer Cluster 2"."T-67.00_CIP_LineOK");
END_REGION

REGION Network 19: BFT 67 Feedback Instrument
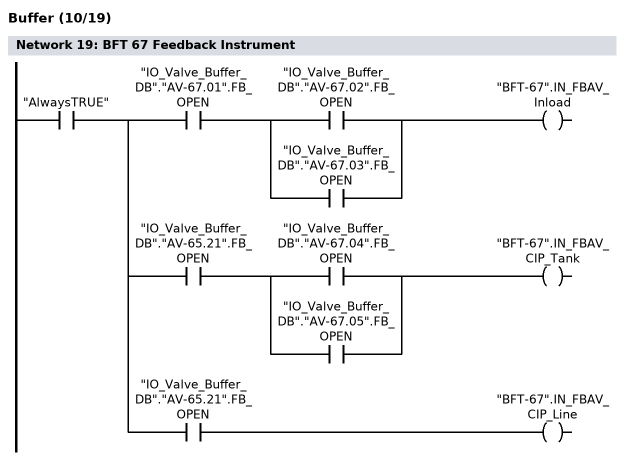
   RUNG wire#powerrail
      Contact( "AlwaysTRUE" )
      wire#w1
      Contact( "IO_Valve_Buffer_DB"."AV-67.01".FB_OPEN )
      wire#w2
      Contact( "IO_Valve_Buffer_DB"."AV-67.02".FB_OPEN )
      wire#w3
      Coil( "BFT-67".IN_FBAV_Inload )
   END_RUNG
   RUNG wire#w2
      Contact( "IO_Valve_Buffer_DB"."AV-67.03".FB_OPEN )
   END_RUNG wire#w3
   RUNG wire#w1
      Contact( "IO_Valve_Buffer_DB"."AV-65.21".FB_OPEN )
      wire#w4
      Contact( "IO_Valve_Buffer_DB"."AV-67.04".FB_OPEN )
      wire#w5
      Coil( "BFT-67".IN_FBAV_CIP_Tank )
   END_RUNG
   RUNG wire#w4
      Contact( "IO_Valve_Buffer_DB"."AV-67.05".FB_OPEN )
   END_RUNG wire#w5
   RUNG wire#w1
      Contact( "IO_Valve_Buffer_DB"."AV-65.21".FB_OPEN )
      Coil( "BFT-67".IN_FBAV_CIP_Line )
   END_RUNG
   // the same network as SCL:
   "BFT-67".IN_FBAV_Inload := "AlwaysTRUE" AND "IO_Valve_Buffer_DB"."AV-67.01".FB_OPEN AND ("IO_Valve_Buffer_DB"."AV-67.02".FB_OPEN OR "IO_Valve_Buffer_DB"."AV-67.03".FB_OPEN);
   "BFT-67".IN_FBAV_CIP_Tank := "AlwaysTRUE" AND "IO_Valve_Buffer_DB"."AV-65.21".FB_OPEN AND ("IO_Valve_Buffer_DB"."AV-67.04".FB_OPEN OR "IO_Valve_Buffer_DB"."AV-67.05".FB_OPEN);
   "BFT-67".IN_FBAV_CIP_Line := "AlwaysTRUE" AND "IO_Valve_Buffer_DB"."AV-65.21".FB_OPEN;
END_REGION

REGION Network 20: BFT 68
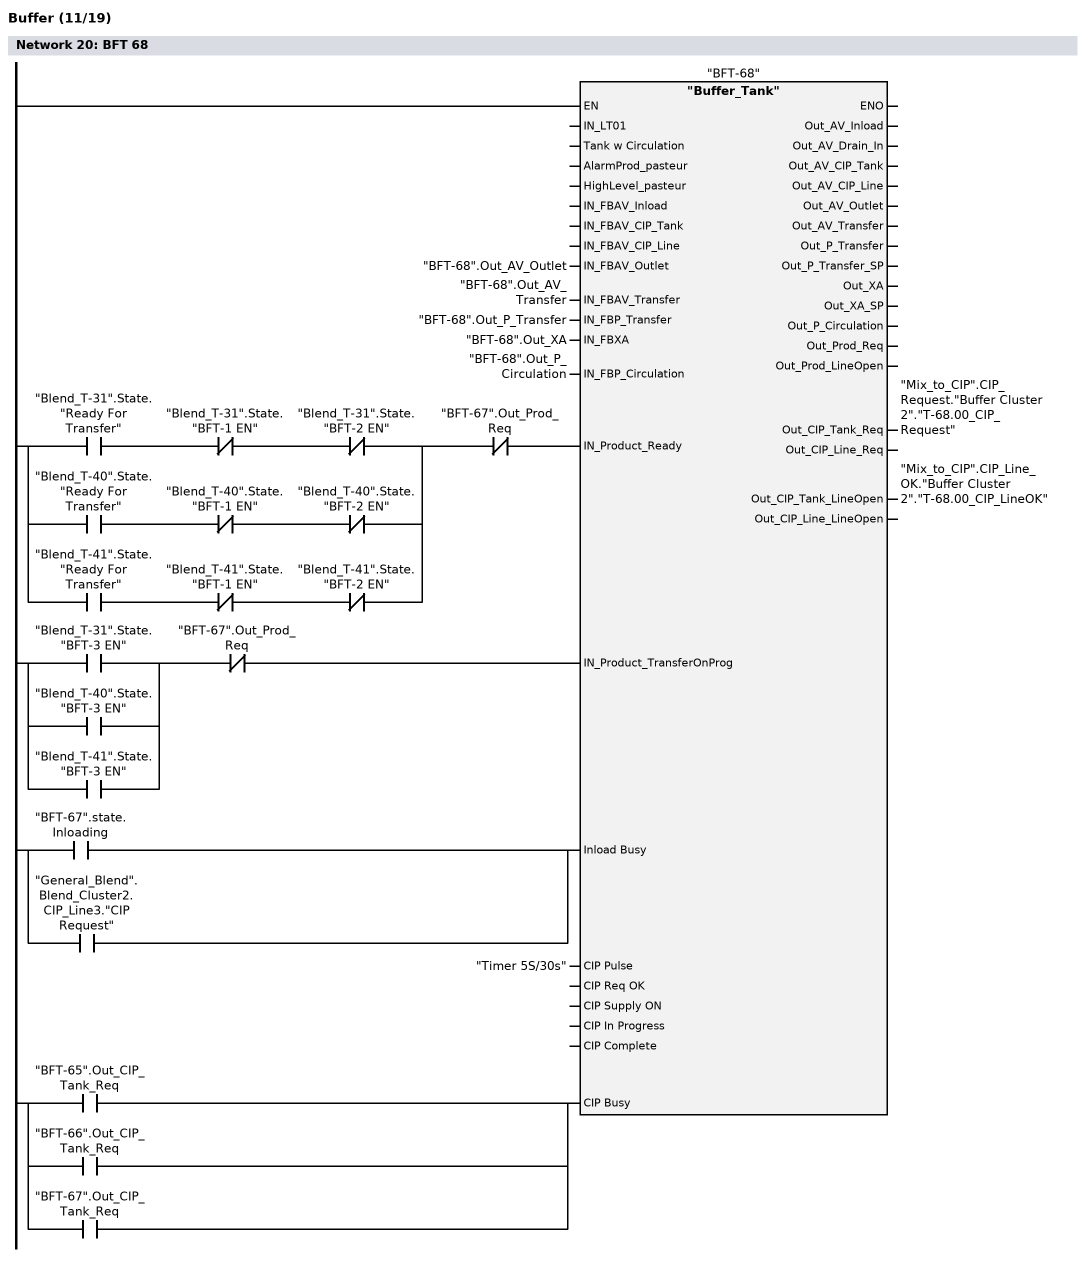
   RUNG wire#powerrail
      "BFT-68"(IN_Product_Ready := wire#w2, IN_Product_TransferOnProg := wire#w4, "Inload Busy" := wire#w5, "CIP Busy" := wire#w6, IN_LT01 :=, "Tank w Circulation" :=, AlarmProd_pasteur :=, HighLevel_pasteur :=, IN_FBAV_Inload :=, IN_FBAV_CIP_Tank :=, IN_FBAV_CIP_Line :=, IN_FBAV_Outlet := "BFT-68".Out_AV_Outlet, IN_FBAV_Transfer := "BFT-68".Out_AV_Transfer, IN_FBP_Transfer := "BFT-68".Out_P_Transfer, IN_FBXA := "BFT-68".Out_XA, IN_FBP_Circulation := "BFT-68".Out_P_Circulation, "CIP Pulse" := "Timer 5S/30s", "CIP Req OK" :=, "CIP Supply ON" :=, "CIP In Progress" :=, "CIP Complete" :=, Out_AV_Inload =>, Out_AV_Drain_In =>, Out_AV_CIP_Tank =>, Out_AV_CIP_Line =>, Out_AV_Outlet =>, Out_AV_Transfer =>, Out_P_Transfer =>, Out_P_Transfer_SP =>, Out_XA =>, Out_XA_SP =>, Out_P_Circulation =>, Out_Prod_Req =>, Out_Prod_LineOpen =>, Out_CIP_Tank_Req => "Mix_to_CIP".CIP_Request."Buffer Cluster 2"."T-68.00_CIP_Request", Out_CIP_Line_Req =>, Out_CIP_Tank_LineOpen => "Mix_to_CIP".CIP_Line_OK."Buffer Cluster 2"."T-68.00_CIP_LineOK", Out_CIP_Line_LineOpen =>)
   END_RUNG
   RUNG wire#powerrail
      Contact( "Blend_T-31".State."Ready For Transfer" )
      I_Contact( "Blend_T-31".State."BFT-1 EN" )
      I_Contact( "Blend_T-31".State."BFT-2 EN" )
      wire#w1
      I_Contact( "BFT-67".Out_Prod_Req )
   END_RUNG wire#w2
   RUNG wire#powerrail
      Contact( "Blend_T-40".State."Ready For Transfer" )
      I_Contact( "Blend_T-40".State."BFT-1 EN" )
      I_Contact( "Blend_T-40".State."BFT-2 EN" )
   END_RUNG wire#w1
   RUNG wire#powerrail
      Contact( "Blend_T-41".State."Ready For Transfer" )
      I_Contact( "Blend_T-41".State."BFT-1 EN" )
      I_Contact( "Blend_T-41".State."BFT-2 EN" )
   END_RUNG wire#w1
   RUNG wire#powerrail
      Contact( "Blend_T-31".State."BFT-3 EN" )
      wire#w3
      I_Contact( "BFT-67".Out_Prod_Req )
   END_RUNG wire#w4
   RUNG wire#powerrail
      Contact( "Blend_T-40".State."BFT-3 EN" )
   END_RUNG wire#w3
   RUNG wire#powerrail
      Contact( "Blend_T-41".State."BFT-3 EN" )
   END_RUNG wire#w3
   RUNG wire#powerrail
      Contact( "BFT-67".state.Inloading )
   END_RUNG wire#w5
   RUNG wire#powerrail
      Contact( "General_Blend".Blend_Cluster2.CIP_Line3."CIP Request" )
   END_RUNG wire#w5
   RUNG wire#powerrail
      Contact( "BFT-65".Out_CIP_Tank_Req )
   END_RUNG wire#w6
   RUNG wire#powerrail
      Contact( "BFT-66".Out_CIP_Tank_Req )
   END_RUNG wire#w6
   RUNG wire#powerrail
      Contact( "BFT-67".Out_CIP_Tank_Req )
   END_RUNG wire#w6
   // the same network as SCL:
   "BFT-68"(IN_FBAV_Outlet := "BFT-68".Out_AV_Outlet,   // "Buffer_Tank"
            IN_FBAV_Transfer := "BFT-68".Out_AV_Transfer,
            IN_FBP_Transfer := "BFT-68".Out_P_Transfer,
            IN_FBXA := "BFT-68".Out_XA,
            IN_FBP_Circulation := "BFT-68".Out_P_Circulation,
            IN_Product_Ready := (("Blend_T-31".State."Ready For Transfer" AND NOT "Blend_T-31".State."BFT-1 EN" AND NOT "Blend_T-31".State."BFT-2 EN") OR ("Blend_T-40".State."Ready For Transfer" AND NOT "Blend_T-40".State."BFT-1 EN" AND NOT "Blend_T-40".State."BFT-2 EN") OR ("Blend_T-41".State."Ready For Transfer" AND NOT "Blend_T-41".State."BFT-1 EN" AND NOT "Blend_T-41".State."BFT-2 EN")) AND NOT "BFT-67".Out_Prod_Req,
            IN_Product_TransferOnProg := ("Blend_T-31".State."BFT-3 EN" OR "Blend_T-40".State."BFT-3 EN" OR "Blend_T-41".State."BFT-3 EN") AND NOT "BFT-67".Out_Prod_Req,
            "Inload Busy" := "BFT-67".state.Inloading OR "General_Blend".Blend_Cluster2.CIP_Line3."CIP Request",
            "CIP Pulse" := "Timer 5S/30s",
            "CIP Busy" := "BFT-65".Out_CIP_Tank_Req OR "BFT-66".Out_CIP_Tank_Req OR "BFT-67".Out_CIP_Tank_Req,
            Out_CIP_Tank_Req => "Mix_to_CIP".CIP_Request."Buffer Cluster 2"."T-68.00_CIP_Request",
            Out_CIP_Tank_LineOpen => "Mix_to_CIP".CIP_Line_OK."Buffer Cluster 2"."T-68.00_CIP_LineOK");
END_REGION

REGION Network 21: BFT 68 Feedback Instrument
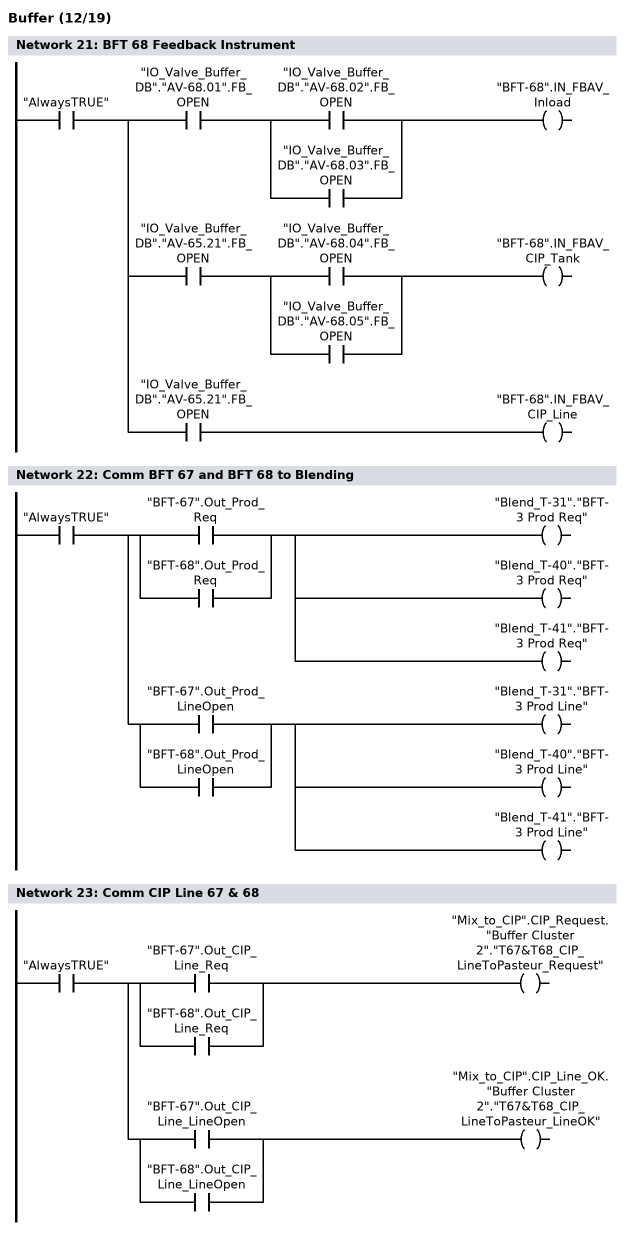
   RUNG wire#powerrail
      Contact( "AlwaysTRUE" )
      wire#w1
      Contact( "IO_Valve_Buffer_DB"."AV-68.01".FB_OPEN )
      wire#w2
      Contact( "IO_Valve_Buffer_DB"."AV-68.02".FB_OPEN )
      wire#w3
      Coil( "BFT-68".IN_FBAV_Inload )
   END_RUNG
   RUNG wire#w2
      Contact( "IO_Valve_Buffer_DB"."AV-68.03".FB_OPEN )
   END_RUNG wire#w3
   RUNG wire#w1
      Contact( "IO_Valve_Buffer_DB"."AV-65.21".FB_OPEN )
      wire#w4
      Contact( "IO_Valve_Buffer_DB"."AV-68.04".FB_OPEN )
      wire#w5
      Coil( "BFT-68".IN_FBAV_CIP_Tank )
   END_RUNG
   RUNG wire#w4
      Contact( "IO_Valve_Buffer_DB"."AV-68.05".FB_OPEN )
   END_RUNG wire#w5
   RUNG wire#w1
      Contact( "IO_Valve_Buffer_DB"."AV-65.21".FB_OPEN )
      Coil( "BFT-68".IN_FBAV_CIP_Line )
   END_RUNG
   // the same network as SCL:
   "BFT-68".IN_FBAV_Inload := "AlwaysTRUE" AND "IO_Valve_Buffer_DB"."AV-68.01".FB_OPEN AND ("IO_Valve_Buffer_DB"."AV-68.02".FB_OPEN OR "IO_Valve_Buffer_DB"."AV-68.03".FB_OPEN);
   "BFT-68".IN_FBAV_CIP_Tank := "AlwaysTRUE" AND "IO_Valve_Buffer_DB"."AV-65.21".FB_OPEN AND ("IO_Valve_Buffer_DB"."AV-68.04".FB_OPEN OR "IO_Valve_Buffer_DB"."AV-68.05".FB_OPEN);
   "BFT-68".IN_FBAV_CIP_Line := "AlwaysTRUE" AND "IO_Valve_Buffer_DB"."AV-65.21".FB_OPEN;
END_REGION

REGION Network 22: Comm BFT 67 and BFT 68 to Blending
   RUNG wire#powerrail
      Contact( "AlwaysTRUE" )
      wire#w1
      Contact( "BFT-67".Out_Prod_Req )
      wire#w2
      Coil( "Blend_T-31"."BFT-3 Prod Req" )
   END_RUNG
   RUNG wire#w1
      Contact( "BFT-68".Out_Prod_Req )
   END_RUNG wire#w2
   RUNG wire#w2
      Coil( "Blend_T-40"."BFT-3 Prod Req" )
   END_RUNG
   RUNG wire#w2
      Coil( "Blend_T-41"."BFT-3 Prod Req" )
   END_RUNG
   RUNG wire#w1
      Contact( "BFT-67".Out_Prod_LineOpen )
      wire#w3
      Coil( "Blend_T-31"."BFT-3 Prod Line" )
   END_RUNG
   RUNG wire#w1
      Contact( "BFT-68".Out_Prod_LineOpen )
   END_RUNG wire#w3
   RUNG wire#w3
      Coil( "Blend_T-40"."BFT-3 Prod Line" )
   END_RUNG
   RUNG wire#w3
      Coil( "Blend_T-41"."BFT-3 Prod Line" )
   END_RUNG
   // the same network as SCL:
   "Blend_T-31"."BFT-3 Prod Req" := "AlwaysTRUE" AND ("BFT-67".Out_Prod_Req OR "BFT-68".Out_Prod_Req);
   "Blend_T-40"."BFT-3 Prod Req" := "Blend_T-31"."BFT-3 Prod Req";
   "Blend_T-41"."BFT-3 Prod Req" := "Blend_T-31"."BFT-3 Prod Req";
   "Blend_T-31"."BFT-3 Prod Line" := "AlwaysTRUE" AND ("BFT-67".Out_Prod_LineOpen OR "BFT-68".Out_Prod_LineOpen);
   "Blend_T-40"."BFT-3 Prod Line" := "Blend_T-31"."BFT-3 Prod Line";
   "Blend_T-41"."BFT-3 Prod Line" := "Blend_T-31"."BFT-3 Prod Line";
END_REGION

REGION Network 23: Comm CIP Line 67 & 68
   RUNG wire#powerrail
      Contact( "AlwaysTRUE" )
      wire#w1
      Contact( "BFT-67".Out_CIP_Line_Req )
      wire#w2
      Coil( "Mix_to_CIP".CIP_Request."Buffer Cluster 2"."T67&T68_CIP_LineToPasteur_Request" )
   END_RUNG
   RUNG wire#w1
      Contact( "BFT-68".Out_CIP_Line_Req )
   END_RUNG wire#w2
   RUNG wire#w1
      Contact( "BFT-67".Out_CIP_Line_LineOpen )
      wire#w3
      Coil( "Mix_to_CIP".CIP_Line_OK."Buffer Cluster 2"."T67&T68_CIP_LineToPasteur_LineOK" )
   END_RUNG
   RUNG wire#w1
      Contact( "BFT-68".Out_CIP_Line_LineOpen )
   END_RUNG wire#w3
   // the same network as SCL:
   "Mix_to_CIP".CIP_Request."Buffer Cluster 2"."T67&T68_CIP_LineToPasteur_Request" := "AlwaysTRUE" AND ("BFT-67".Out_CIP_Line_Req OR "BFT-68".Out_CIP_Line_Req);
   "Mix_to_CIP".CIP_Line_OK."Buffer Cluster 2"."T67&T68_CIP_LineToPasteur_LineOK" := "AlwaysTRUE" AND ("BFT-67".Out_CIP_Line_LineOpen OR "BFT-68".Out_CIP_Line_LineOpen);
END_REGION

REGION Network 25: Comm CIP to BFT 61 Rework 32
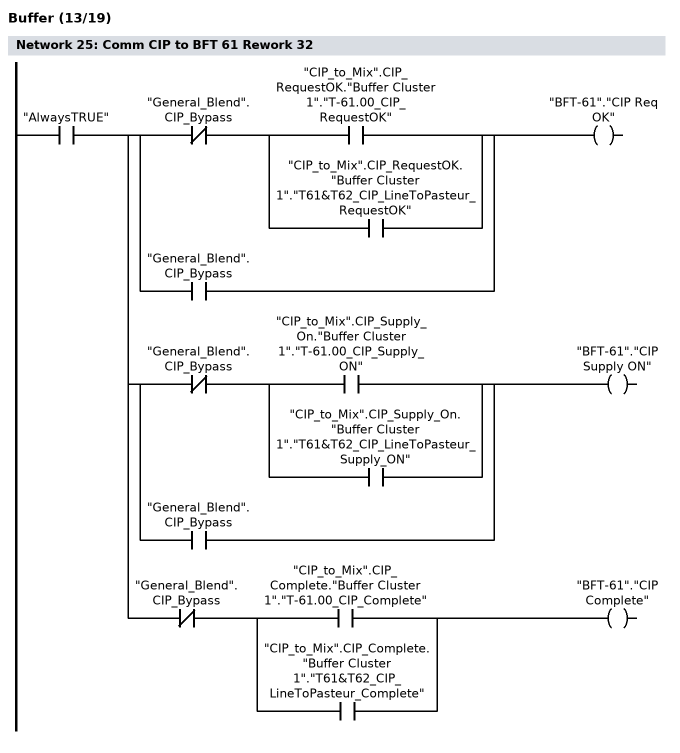
   RUNG wire#powerrail
      Contact( "AlwaysTRUE" )
      wire#w1
      I_Contact( "General_Blend".CIP_Bypass )
      wire#w2
      Contact( "CIP_to_Mix".CIP_RequestOK."Buffer Cluster 1"."T-61.00_CIP_RequestOK" )
      wire#w3
      Coil( "BFT-61"."CIP Req OK" )
   END_RUNG
   RUNG wire#w2
      Contact( "CIP_to_Mix".CIP_RequestOK."Buffer Cluster 1"."T61&T62_CIP_LineToPasteur_RequestOK" )
   END_RUNG wire#w3
   RUNG wire#w1
      Contact( "General_Blend".CIP_Bypass )
   END_RUNG wire#w3
   RUNG wire#w1
      I_Contact( "General_Blend".CIP_Bypass )
      wire#w4
      Contact( "CIP_to_Mix".CIP_Supply_On."Buffer Cluster 1"."T-61.00_CIP_Supply_ON" )
      wire#w5
      Coil( "BFT-61"."CIP Supply ON" )
   END_RUNG
   RUNG wire#w4
      Contact( "CIP_to_Mix".CIP_Supply_On."Buffer Cluster 1"."T61&T62_CIP_LineToPasteur_Supply_ON" )
   END_RUNG wire#w5
   RUNG wire#w1
      Contact( "General_Blend".CIP_Bypass )
   END_RUNG wire#w5
   RUNG wire#w1
      I_Contact( "General_Blend".CIP_Bypass )
      wire#w6
      Contact( "CIP_to_Mix".CIP_Complete."Buffer Cluster 1"."T-61.00_CIP_Complete" )
      wire#w7
      Coil( "BFT-61"."CIP Complete" )
   END_RUNG
   RUNG wire#w6
      Contact( "CIP_to_Mix".CIP_Complete."Buffer Cluster 1"."T61&T62_CIP_LineToPasteur_Complete" )
   END_RUNG wire#w7
   // the same network as SCL:
   "BFT-61"."CIP Req OK" := "AlwaysTRUE" AND ((NOT "General_Blend".CIP_Bypass AND ("CIP_to_Mix".CIP_RequestOK."Buffer Cluster 1"."T-61.00_CIP_RequestOK" OR "CIP_to_Mix".CIP_RequestOK."Buffer Cluster 1"."T61&T62_CIP_LineToPasteur_RequestOK")) OR "General_Blend".CIP_Bypass);
   "BFT-61"."CIP Supply ON" := "AlwaysTRUE" AND ((NOT "General_Blend".CIP_Bypass AND ("CIP_to_Mix".CIP_Supply_On."Buffer Cluster 1"."T-61.00_CIP_Supply_ON" OR "CIP_to_Mix".CIP_Supply_On."Buffer Cluster 1"."T61&T62_CIP_LineToPasteur_Supply_ON")) OR "General_Blend".CIP_Bypass);
   "BFT-61"."CIP Complete" := "AlwaysTRUE" AND NOT "General_Blend".CIP_Bypass AND ("CIP_to_Mix".CIP_Complete."Buffer Cluster 1"."T-61.00_CIP_Complete" OR "CIP_to_Mix".CIP_Complete."Buffer Cluster 1"."T61&T62_CIP_LineToPasteur_Complete");
END_REGION

REGION Network 26: Comm CIP to BFT 64 Rework 22
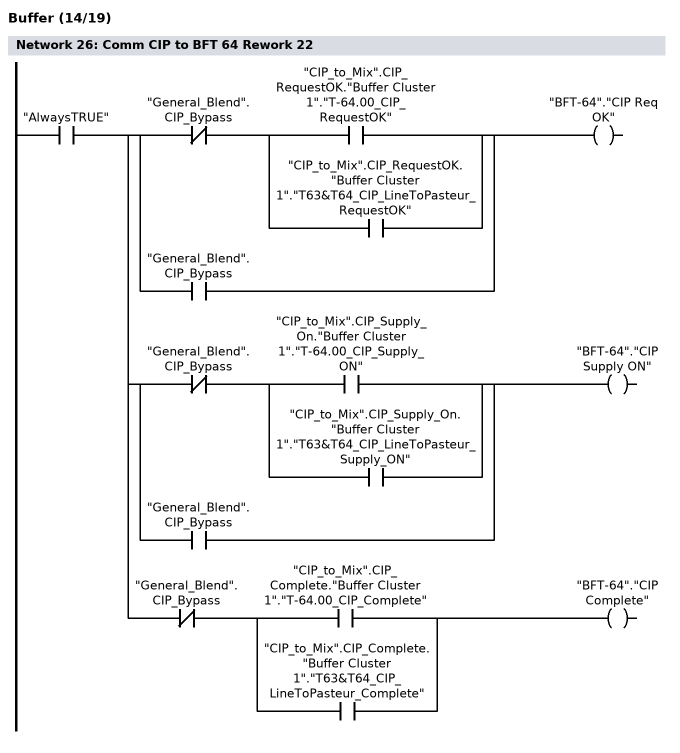
   RUNG wire#powerrail
      Contact( "AlwaysTRUE" )
      wire#w1
      I_Contact( "General_Blend".CIP_Bypass )
      wire#w2
      Contact( "CIP_to_Mix".CIP_RequestOK."Buffer Cluster 1"."T-64.00_CIP_RequestOK" )
      wire#w3
      Coil( "BFT-64"."CIP Req OK" )
   END_RUNG
   RUNG wire#w2
      Contact( "CIP_to_Mix".CIP_RequestOK."Buffer Cluster 1"."T63&T64_CIP_LineToPasteur_RequestOK" )
   END_RUNG wire#w3
   RUNG wire#w1
      Contact( "General_Blend".CIP_Bypass )
   END_RUNG wire#w3
   RUNG wire#w1
      I_Contact( "General_Blend".CIP_Bypass )
      wire#w4
      Contact( "CIP_to_Mix".CIP_Supply_On."Buffer Cluster 1"."T-64.00_CIP_Supply_ON" )
      wire#w5
      Coil( "BFT-64"."CIP Supply ON" )
   END_RUNG
   RUNG wire#w4
      Contact( "CIP_to_Mix".CIP_Supply_On."Buffer Cluster 1"."T63&T64_CIP_LineToPasteur_Supply_ON" )
   END_RUNG wire#w5
   RUNG wire#w1
      Contact( "General_Blend".CIP_Bypass )
   END_RUNG wire#w5
   RUNG wire#w1
      I_Contact( "General_Blend".CIP_Bypass )
      wire#w6
      Contact( "CIP_to_Mix".CIP_Complete."Buffer Cluster 1"."T-64.00_CIP_Complete" )
      wire#w7
      Coil( "BFT-64"."CIP Complete" )
   END_RUNG
   RUNG wire#w6
      Contact( "CIP_to_Mix".CIP_Complete."Buffer Cluster 1"."T63&T64_CIP_LineToPasteur_Complete" )
   END_RUNG wire#w7
   // the same network as SCL:
   "BFT-64"."CIP Req OK" := "AlwaysTRUE" AND ((NOT "General_Blend".CIP_Bypass AND ("CIP_to_Mix".CIP_RequestOK."Buffer Cluster 1"."T-64.00_CIP_RequestOK" OR "CIP_to_Mix".CIP_RequestOK."Buffer Cluster 1"."T63&T64_CIP_LineToPasteur_RequestOK")) OR "General_Blend".CIP_Bypass);
   "BFT-64"."CIP Supply ON" := "AlwaysTRUE" AND ((NOT "General_Blend".CIP_Bypass AND ("CIP_to_Mix".CIP_Supply_On."Buffer Cluster 1"."T-64.00_CIP_Supply_ON" OR "CIP_to_Mix".CIP_Supply_On."Buffer Cluster 1"."T63&T64_CIP_LineToPasteur_Supply_ON")) OR "General_Blend".CIP_Bypass);
   "BFT-64"."CIP Complete" := "AlwaysTRUE" AND NOT "General_Blend".CIP_Bypass AND ("CIP_to_Mix".CIP_Complete."Buffer Cluster 1"."T-64.00_CIP_Complete" OR "CIP_to_Mix".CIP_Complete."Buffer Cluster 1"."T63&T64_CIP_LineToPasteur_Complete");
END_REGION

REGION Network 27: Comm CIP to BFT 65
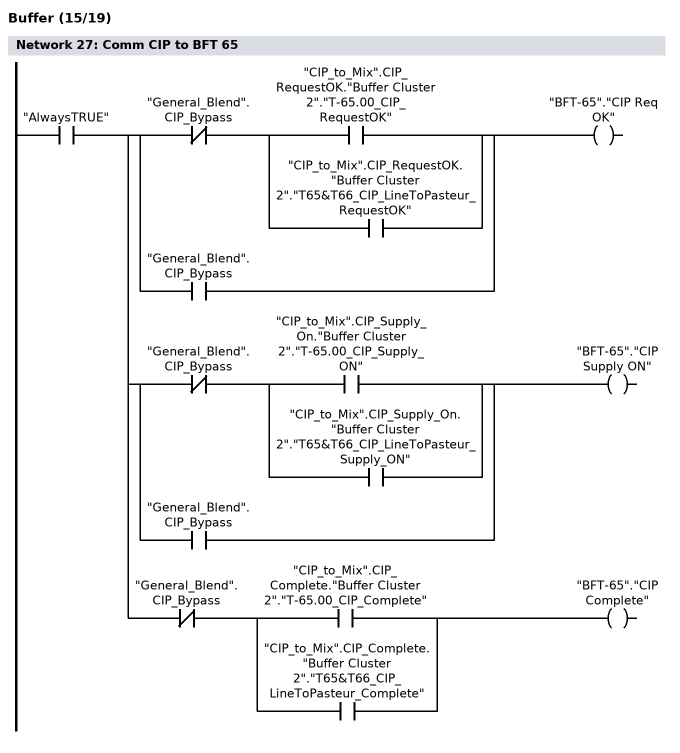
   RUNG wire#powerrail
      Contact( "AlwaysTRUE" )
      wire#w1
      I_Contact( "General_Blend".CIP_Bypass )
      wire#w2
      Contact( "CIP_to_Mix".CIP_RequestOK."Buffer Cluster 2"."T-65.00_CIP_RequestOK" )
      wire#w3
      Coil( "BFT-65"."CIP Req OK" )
   END_RUNG
   RUNG wire#w2
      Contact( "CIP_to_Mix".CIP_RequestOK."Buffer Cluster 2"."T65&T66_CIP_LineToPasteur_RequestOK" )
   END_RUNG wire#w3
   RUNG wire#w1
      Contact( "General_Blend".CIP_Bypass )
   END_RUNG wire#w3
   RUNG wire#w1
      I_Contact( "General_Blend".CIP_Bypass )
      wire#w4
      Contact( "CIP_to_Mix".CIP_Supply_On."Buffer Cluster 2"."T-65.00_CIP_Supply_ON" )
      wire#w5
      Coil( "BFT-65"."CIP Supply ON" )
   END_RUNG
   RUNG wire#w4
      Contact( "CIP_to_Mix".CIP_Supply_On."Buffer Cluster 2"."T65&T66_CIP_LineToPasteur_Supply_ON" )
   END_RUNG wire#w5
   RUNG wire#w1
      Contact( "General_Blend".CIP_Bypass )
   END_RUNG wire#w5
   RUNG wire#w1
      I_Contact( "General_Blend".CIP_Bypass )
      wire#w6
      Contact( "CIP_to_Mix".CIP_Complete."Buffer Cluster 2"."T-65.00_CIP_Complete" )
      wire#w7
      Coil( "BFT-65"."CIP Complete" )
   END_RUNG
   RUNG wire#w6
      Contact( "CIP_to_Mix".CIP_Complete."Buffer Cluster 2"."T65&T66_CIP_LineToPasteur_Complete" )
   END_RUNG wire#w7
   // the same network as SCL:
   "BFT-65"."CIP Req OK" := "AlwaysTRUE" AND ((NOT "General_Blend".CIP_Bypass AND ("CIP_to_Mix".CIP_RequestOK."Buffer Cluster 2"."T-65.00_CIP_RequestOK" OR "CIP_to_Mix".CIP_RequestOK."Buffer Cluster 2"."T65&T66_CIP_LineToPasteur_RequestOK")) OR "General_Blend".CIP_Bypass);
   "BFT-65"."CIP Supply ON" := "AlwaysTRUE" AND ((NOT "General_Blend".CIP_Bypass AND ("CIP_to_Mix".CIP_Supply_On."Buffer Cluster 2"."T-65.00_CIP_Supply_ON" OR "CIP_to_Mix".CIP_Supply_On."Buffer Cluster 2"."T65&T66_CIP_LineToPasteur_Supply_ON")) OR "General_Blend".CIP_Bypass);
   "BFT-65"."CIP Complete" := "AlwaysTRUE" AND NOT "General_Blend".CIP_Bypass AND ("CIP_to_Mix".CIP_Complete."Buffer Cluster 2"."T-65.00_CIP_Complete" OR "CIP_to_Mix".CIP_Complete."Buffer Cluster 2"."T65&T66_CIP_LineToPasteur_Complete");
END_REGION

REGION Network 28: Comm CIP to BFT 66
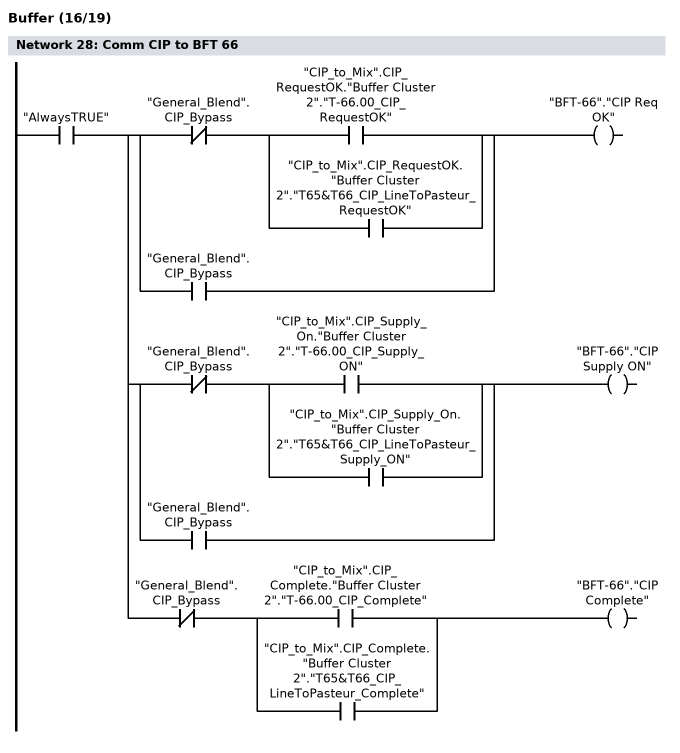
   RUNG wire#powerrail
      Contact( "AlwaysTRUE" )
      wire#w1
      I_Contact( "General_Blend".CIP_Bypass )
      wire#w2
      Contact( "CIP_to_Mix".CIP_RequestOK."Buffer Cluster 2"."T-66.00_CIP_RequestOK" )
      wire#w3
      Coil( "BFT-66"."CIP Req OK" )
   END_RUNG
   RUNG wire#w2
      Contact( "CIP_to_Mix".CIP_RequestOK."Buffer Cluster 2"."T65&T66_CIP_LineToPasteur_RequestOK" )
   END_RUNG wire#w3
   RUNG wire#w1
      Contact( "General_Blend".CIP_Bypass )
   END_RUNG wire#w3
   RUNG wire#w1
      I_Contact( "General_Blend".CIP_Bypass )
      wire#w4
      Contact( "CIP_to_Mix".CIP_Supply_On."Buffer Cluster 2"."T-66.00_CIP_Supply_ON" )
      wire#w5
      Coil( "BFT-66"."CIP Supply ON" )
   END_RUNG
   RUNG wire#w4
      Contact( "CIP_to_Mix".CIP_Supply_On."Buffer Cluster 2"."T65&T66_CIP_LineToPasteur_Supply_ON" )
   END_RUNG wire#w5
   RUNG wire#w1
      Contact( "General_Blend".CIP_Bypass )
   END_RUNG wire#w5
   RUNG wire#w1
      I_Contact( "General_Blend".CIP_Bypass )
      wire#w6
      Contact( "CIP_to_Mix".CIP_Complete."Buffer Cluster 2"."T-66.00_CIP_Complete" )
      wire#w7
      Coil( "BFT-66"."CIP Complete" )
   END_RUNG
   RUNG wire#w6
      Contact( "CIP_to_Mix".CIP_Complete."Buffer Cluster 2"."T65&T66_CIP_LineToPasteur_Complete" )
   END_RUNG wire#w7
   // the same network as SCL:
   "BFT-66"."CIP Req OK" := "AlwaysTRUE" AND ((NOT "General_Blend".CIP_Bypass AND ("CIP_to_Mix".CIP_RequestOK."Buffer Cluster 2"."T-66.00_CIP_RequestOK" OR "CIP_to_Mix".CIP_RequestOK."Buffer Cluster 2"."T65&T66_CIP_LineToPasteur_RequestOK")) OR "General_Blend".CIP_Bypass);
   "BFT-66"."CIP Supply ON" := "AlwaysTRUE" AND ((NOT "General_Blend".CIP_Bypass AND ("CIP_to_Mix".CIP_Supply_On."Buffer Cluster 2"."T-66.00_CIP_Supply_ON" OR "CIP_to_Mix".CIP_Supply_On."Buffer Cluster 2"."T65&T66_CIP_LineToPasteur_Supply_ON")) OR "General_Blend".CIP_Bypass);
   "BFT-66"."CIP Complete" := "AlwaysTRUE" AND NOT "General_Blend".CIP_Bypass AND ("CIP_to_Mix".CIP_Complete."Buffer Cluster 2"."T-66.00_CIP_Complete" OR "CIP_to_Mix".CIP_Complete."Buffer Cluster 2"."T65&T66_CIP_LineToPasteur_Complete");
END_REGION

REGION Network 29: Comm CIP to BFT 67
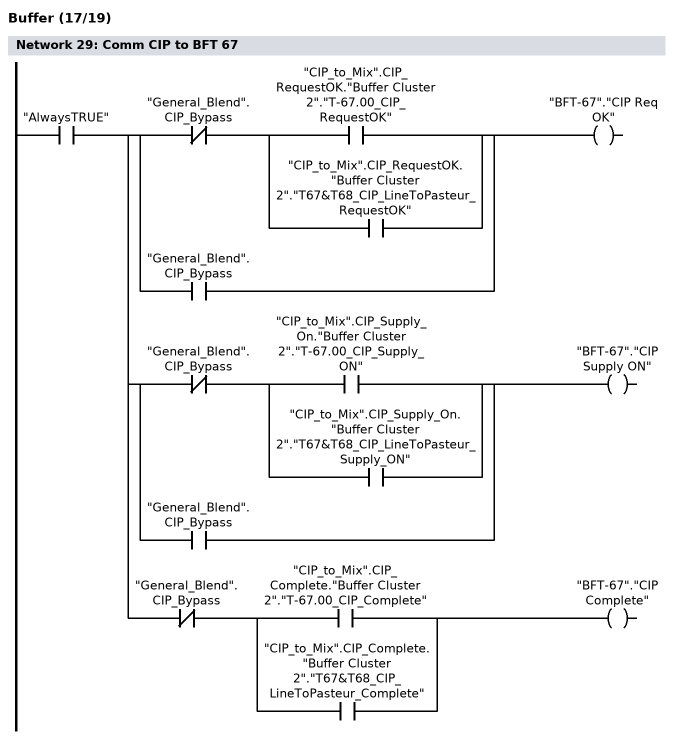
   RUNG wire#powerrail
      Contact( "AlwaysTRUE" )
      wire#w1
      I_Contact( "General_Blend".CIP_Bypass )
      wire#w2
      Contact( "CIP_to_Mix".CIP_RequestOK."Buffer Cluster 2"."T-67.00_CIP_RequestOK" )
      wire#w3
      Coil( "BFT-67"."CIP Req OK" )
   END_RUNG
   RUNG wire#w2
      Contact( "CIP_to_Mix".CIP_RequestOK."Buffer Cluster 2"."T67&T68_CIP_LineToPasteur_RequestOK" )
   END_RUNG wire#w3
   RUNG wire#w1
      Contact( "General_Blend".CIP_Bypass )
   END_RUNG wire#w3
   RUNG wire#w1
      I_Contact( "General_Blend".CIP_Bypass )
      wire#w4
      Contact( "CIP_to_Mix".CIP_Supply_On."Buffer Cluster 2"."T-67.00_CIP_Supply_ON" )
      wire#w5
      Coil( "BFT-67"."CIP Supply ON" )
   END_RUNG
   RUNG wire#w4
      Contact( "CIP_to_Mix".CIP_Supply_On."Buffer Cluster 2"."T67&T68_CIP_LineToPasteur_Supply_ON" )
   END_RUNG wire#w5
   RUNG wire#w1
      Contact( "General_Blend".CIP_Bypass )
   END_RUNG wire#w5
   RUNG wire#w1
      I_Contact( "General_Blend".CIP_Bypass )
      wire#w6
      Contact( "CIP_to_Mix".CIP_Complete."Buffer Cluster 2"."T-67.00_CIP_Complete" )
      wire#w7
      Coil( "BFT-67"."CIP Complete" )
   END_RUNG
   RUNG wire#w6
      Contact( "CIP_to_Mix".CIP_Complete."Buffer Cluster 2"."T67&T68_CIP_LineToPasteur_Complete" )
   END_RUNG wire#w7
   // the same network as SCL:
   "BFT-67"."CIP Req OK" := "AlwaysTRUE" AND ((NOT "General_Blend".CIP_Bypass AND ("CIP_to_Mix".CIP_RequestOK."Buffer Cluster 2"."T-67.00_CIP_RequestOK" OR "CIP_to_Mix".CIP_RequestOK."Buffer Cluster 2"."T67&T68_CIP_LineToPasteur_RequestOK")) OR "General_Blend".CIP_Bypass);
   "BFT-67"."CIP Supply ON" := "AlwaysTRUE" AND ((NOT "General_Blend".CIP_Bypass AND ("CIP_to_Mix".CIP_Supply_On."Buffer Cluster 2"."T-67.00_CIP_Supply_ON" OR "CIP_to_Mix".CIP_Supply_On."Buffer Cluster 2"."T67&T68_CIP_LineToPasteur_Supply_ON")) OR "General_Blend".CIP_Bypass);
   "BFT-67"."CIP Complete" := "AlwaysTRUE" AND NOT "General_Blend".CIP_Bypass AND ("CIP_to_Mix".CIP_Complete."Buffer Cluster 2"."T-67.00_CIP_Complete" OR "CIP_to_Mix".CIP_Complete."Buffer Cluster 2"."T67&T68_CIP_LineToPasteur_Complete");
END_REGION

REGION Network 30: Comm CIP to BFT 68
